IF bErrorBlinking THEN
	Error := FALSE;
END_IF

IF NOT Execute THEN
	bErrorBlinking := FALSE;
	tonErrorResetDelay.IN := FALSE;
	eSTATE:=STATE_RESETTING;
END_IF
END_METHOD

METHOD  M_STATE_EXECUTING
VAR_INPUT
END_VAR
VAR_INST
	bMoveConveyorForward : BOOL;
	bMoveConveyorBackrward : BOOL;
END_VAR

VAR
	bCylinderCheck : BOOL := TRUE;
END_VAR
Busy :=TRUE;
SensorOnConveyor := INPUT.bDifferentSizeCV_BoxDetect5_Sensor;

// ============================================================
// (A) Step 切換 → Timer 完整歸零 (Fix 1)
// ============================================================
IF uiExecutingStep <> uiExecutingStep_Last THEN
	tonTimeOut(IN:=FALSE);
	tonTimeDelay(IN:=FALSE);
	tonLeaveDebounce(IN:=FALSE);
	uiExecutingStep_Last := uiExecutingStep;
END_IF

// ============================================================
// (B) TurnTable Interlock (Fix 3)
// Place 下爪區間 (2200~2499) 與 TT 偵測區間 (2600) 期間
// TurnTable 不可移動 (pick 階段在 I5 conveyor,與 TT 無關)
// ============================================================
IF (uiExecutingStep >= 2200 AND uiExecutingStep <= 2499)
OR (uiExecutingStep = 2600)
THEN
	IF arAxisCtrl_gb[AxisNo.TurnTable].Admin.Axis.Status.Moving THEN
		_Error := TRUE;
		uiResumeStep := uiExecutingStep;
		strStatus := M_FormatManagedStatus(
			AlarmId := GVL_ErrorCode.GC_ALARM_ALC_OUTROBOT_EMPTY,
			InnerMessage := GVL_ErrorCode.GC_MSG_0174);
		Status := strStatus;
		Error := TRUE;
	END_IF
END_IF

// ============================================================
// (C) Pause 處理 (Fix 4) - 僅在「安全 step」生效
// ============================================================
bCanPause :=
	   uiExecutingStep = 0
	OR uiExecutingStep = 100
	OR uiExecutingStep = 200
	OR uiExecutingStep = 1000
	OR uiExecutingStep = 1100
	OR uiExecutingStep = 1400
	OR uiExecutingStep = 1900
	OR uiExecutingStep = 2000
	OR uiExecutingStep = 2100
	OR uiExecutingStep = 2500;

// Pause 釋放邊緣 → 強制 timer 歸零 (避免 release 瞬間誤判)
IF bPauseLast AND NOT Pause THEN
	tonTimeOut(IN:=FALSE);
	tonTimeDelay(IN:=FALSE);
	tonLeaveDebounce(IN:=FALSE);
END_IF
bPauseLast := Pause;

IF Pause AND bCanPause THEN
	bMoveConveyorForward := FALSE;
	bMoveConveyorBackrward := FALSE;
	IF __ISVALIDREF(ConveyorMotor) THEN
		ConveyorMotor.M_MotorStop();
	END_IF
	tonTimeOut(IN:=FALSE);
	tonTimeDelay(IN:=FALSE);
	tonLeaveDebounce(IN:=FALSE);
	Busy := TRUE;
	RETURN;
END_IF

// ============================================================
// Conveyor 連續控制 (沿用既有 latched flag)
// ============================================================
IF bMoveConveyorForward THEN
	IF NOT ConveyorMotor.InBackWard THEN
		ConveyorMotor.M_MoveForward();
	END_IF
END_IF
IF bMoveConveyorBackrward THEN
	IF NOT ConveyorMotor.InForWard THEN
		ConveyorMotor.M_MoveBackward();
	END_IF
END_IF

CASE uiExecutingStep OF

0: //Entry - VAR_INST reset + working conditions
	// VAR_INST 私有給本 method,DORMANT 看不到,必須在此 reset
	bMoveConveyorForward := FALSE;
	bMoveConveyorBackrward := FALSE;

	IF GVL_Machine.PackTags[UnitNo.Allocate].Status.UnitModeCurrent <> E_UnitMode.Auto THEN
		strStatus := 'Not in Auto mode';
		_UniqueErrorCode := 'E_NOT_AUTO_MODE';
		_Error := TRUE;
	ELSIF bResumeEnabled AND uiResumeStep > 0 THEN
		// 續做模式: M_GetWorkingConditions 重新取 clamping info (可能已改)
		IF M_GetWorkingConditions() THEN
			M_RecoveryAllObjects();
			// Safety: 若仍夾著箱,強制走 placing 流程 (絕不能回 pick 再抓一個)
			IF bClipHasBox[0] OR bClipHasBox[1] THEN
				IF bClipHasBox[0] THEN
					iWorkingIndex := 0;
				ELSE
					iWorkingIndex := 1;
				END_IF
				// 對齊 pick/place 進度: 未握箱的側視為「無須再處理」
				bPickedA := UseA;
				bPickedB := UseB;
				bPlacedA := UseA AND NOT bClipHasBox[0];
				bPlacedB := UseB AND NOT bClipHasBox[1];
				uiExecutingStep := 2000;	// 直接進 placing (會重檢 TT 角度)
			ELSE
				uiExecutingStep := M_GetResumeEntryStep(uiErrorStep:=uiResumeStep);
			END_IF
			bResumeEnabled := FALSE;
			uiResumeStep := 0;
		ELSE
			_Error := TRUE;
		END_IF
	ELSE
		// 正常啟動: DORMANT 已 reset 所有 FB-level flag,此處讀 input + recover 物件
		IF M_GetWorkingConditions() THEN
			M_RecoveryAllObjects();
			uiExecutingStep := 100;
		ELSE
			_Error := TRUE;
		END_IF
	END_IF

100: //Check command
	IF __ISVALIDREF(PressCylinderOnI5) THEN
		IF PressCylinderOnI5.xError THEN
			PressCylinderOnI5.M_Reset();
		ELSE
			PressCylinderOnI5.M_Retract();
		END_IF
	END_IF

	IF M_CheckCommand() THEN
		uiExecutingStep:=200;
	ELSE
		_Error := TRUE;
	END_IF

200: // Check no boxes on TurnTable (殘箱 → 不可續做)
	IF (UseA AND INPUT.bTurnTable_R1Detect_Sensor) OR (UseB AND INPUT.bTurnTable_R2Detect_Sensor) THEN
		_Abort:=TRUE;
		uiResumeStep := 0;	// 殘箱錯誤禁止續做
		strStatus := M_FormatManagedStatus(
			AlarmId := GVL_ErrorCode.GC_ALARM_ALC_OUTROBOT_EMPTY,
			InnerMessage := GVL_ErrorCode.GC_MSG_0012);
		Status := strStatus;
		Error := TRUE;
	ELSE
		IF UseA THEN
			iWorkingIndex :=0;
		ELSE
			iWorkingIndex :=1;
		END_IF
		uiExecutingStep:=1000;
	END_IF

1000: // Move conveyor forward + send OutRobot to picking pos
	bMoveConveyorForward:=TRUE;
	arAxisCtrl_gb[AxisNo.OutRobot_X].PosMode.Position := PickingPos[iWorkingIndex].X_Pos;
	arAxisCtrl_gb[AxisNo.OutRobot_Y].PosMode.Position := PickingPos[iWorkingIndex].Y_Pos;
	IF ConveyorMotor.InForWard THEN
		uiExecutingStep:=1100;
	END_IF

1100: // Wait box arriving sensor (1s debounce)
	tonTimeDelay(IN:=SensorOnConveyor, PT:=T#1S);
	IF tonTimeDelay.Q THEN
		uiExecutingStep:=1200;
	ELSE
		tonTimeOut(IN:=TRUE, PT:=T#15S);
		IF tonTimeOut.Q THEN
			_Abort := TRUE;
			uiResumeStep := uiExecutingStep;
			strStatus := M_FormatManagedStatus(
				AlarmId := GVL_ErrorCode.GC_ALARM_ALC_OUTROBOT_EMPTY,
				InnerMessage := GVL_ErrorCode.GC_MSG_0088);
			Status := strStatus;
			Error := TRUE;
		END_IF
	END_IF

1200: // (預留) Press second box - 目前不執行,直接 fall-through
	uiExecutingStep:=1300;

1300: // Stop conveyor
	ConveyorMotor.M_MotorStop();
	bMoveConveyorForward:=FALSE;
	bMoveConveyorBackrward:=FALSE;
	IF ConveyorMotor.InStopped THEN
		uiExecutingStep:=1400;
	END_IF

1400: // Wait OutRobot XY arrive (pick)
	IF (arAxisStatus_gb[AxisNo.OutRobot_X].Admin._OpModeAck = ModePosAbs AND arAxisStatus_gb[AxisNo.OutRobot_X].Admin.CmdDone)
	AND (arAxisStatus_gb[AxisNo.OutRobot_Y].Admin._OpModeAck = ModePosAbs AND arAxisStatus_gb[AxisNo.OutRobot_Y].Admin.CmdDone)
	THEN
		uiExecutingStep:=1500;
	ELSE
		tonTimeOut(IN:=TRUE, PT:=T#15S);
		IF tonTimeOut.Q THEN
			_Error := TRUE;
			uiResumeStep := uiExecutingStep;
			strStatus := M_FormatManagedStatus(
				AlarmId := GVL_ErrorCode.GC_ALARM_ALC_OUTROBOT_EMPTY,
				InnerMessage := GVL_ErrorCode.GC_MSG_0083);
			Status := strStatus;
			Error := TRUE;
		END_IF
	END_IF

1500: // Clip down (pick) - Fix 2: 下爪前位置再確認
	IF NOT M_IsOutRobotAtPos(TargetPos:=PickingPos[iWorkingIndex]) THEN
		_Error := TRUE;
		uiResumeStep := uiExecutingStep;
		strStatus := M_FormatManagedStatus(
			AlarmId := GVL_ErrorCode.GC_ALARM_ALC_OUTROBOT_EMPTY,
			InnerMessage := GVL_ErrorCode.GC_MSG_0172);
		Status := strStatus;
		Error := TRUE;
	ELSE
		// Sync 對稱化 (S1/S2): sync 時兩爪同動同檢查
		IF bSyncPick THEN
			Cylinders[0].M_Extend();
			Cylinders[1].M_Extend();
			bCylinderCheck := Cylinders[0].InFrontPosition AND Cylinders[1].InFrontPosition;
		ELSE
			Cylinders[iWorkingIndex].M_Extend();
			bCylinderCheck := Cylinders[iWorkingIndex].InFrontPosition;
		END_IF
		IF bCylinderCheck THEN
			uiExecutingStep:=1700;
		ELSE
			tonTimeOut(IN:=TRUE, PT:=T#15S);
			IF tonTimeOut.Q THEN
				_Abort := TRUE;
				uiResumeStep := uiExecutingStep;
				strStatus := M_FormatManagedStatus(
					AlarmId := GVL_ErrorCode.GC_ALARM_ALC_OUTROBOT_EMPTY,
					InnerMessage := GVL_ErrorCode.GC_MSG_0048);
				Status := strStatus;
				Error := TRUE;
			END_IF
		END_IF
	END_IF

1700: // Clip close (pick)
	IF bSyncPick THEN
		Clips[0].M_Extend();
		Clips[1].M_Extend();
		bCylinderCheck := Clips[0].InFrontPosition AND Clips[1].InFrontPosition;
	ELSE
		Clips[iWorkingIndex].M_Extend();
		bCylinderCheck := Clips[iWorkingIndex].InFrontPosition;
	END_IF
	IF bCylinderCheck THEN
		// Safety: 標記夾到箱 (sync 時兩爪都標)
		IF bSyncPick THEN
			bClipHasBox[0] := TRUE;
			bClipHasBox[1] := TRUE;
		ELSE
			bClipHasBox[iWorkingIndex] := TRUE;
		END_IF
		uiExecutingStep:=1800;
	ELSE
		tonTimeOut(IN:=TRUE, PT:=T#15S);
		IF tonTimeOut.Q THEN
			_Abort := TRUE;
			uiResumeStep := uiExecutingStep;
			strStatus := M_FormatManagedStatus(
				AlarmId := GVL_ErrorCode.GC_ALARM_ALC_OUTROBOT_EMPTY,
				InnerMessage := GVL_ErrorCode.GC_MSG_0026);
			Status := strStatus;
			Error := TRUE;
		END_IF
	END_IF

1800: // Clip up (pick)
	IF bSyncPick THEN
		Cylinders[0].M_Retract();
		Cylinders[1].M_Retract();
		bCylinderCheck := Cylinders[0].InRearPosition AND Cylinders[1].InRearPosition;
	ELSE
		Cylinders[iWorkingIndex].M_Retract();
		bCylinderCheck := Cylinders[iWorkingIndex].InRearPosition;
	END_IF
	IF bCylinderCheck THEN
		uiExecutingStep:=1850;
	ELSE
		tonTimeOut(IN:=TRUE, PT:=T#15S);
		IF tonTimeOut.Q THEN
			_Abort := TRUE;
			uiResumeStep := uiExecutingStep;
			strStatus := M_FormatManagedStatus(
				AlarmId := GVL_ErrorCode.GC_ALARM_ALC_OUTROBOT_EMPTY,
				InnerMessage := GVL_ErrorCode.GC_MSG_0050);
			Status := strStatus;
			Error := TRUE;
		END_IF
	END_IF

1850: // Confirm box left conveyor sensor
	// ============================================================
	// TEMP (2026-04-30): A、B 兩爪皆暫時跳過離開檢查
	// 原因: conveyor sensor (BoxDetect5) 只能反映 conveyor 上有無箱,
	//       無法保證箱真的被夾在爪上。A 原本就跳過 (避免上游補料壓
	//       sensor 誤判), B 因相同顧慮也暫時不檢查。
	// 復原條件: 爪上加裝 box-detect sensor,或上游補料時序確認後。
	// 復原方式: 移除本無條件跳過區塊,還原下方 (* *) 內的原邏輯。
	// ============================================================
	tonLeaveDebounce(IN:=FALSE, PT:=T#1S);
	tonTimeOut(IN:=FALSE, PT:=T#15S);
	IF __ISVALIDREF(PressCylinderOnI5) THEN
		PressCylinderOnI5.M_Retract();
	END_IF
	uiExecutingStep:=1900;

	(* ---- 原離開檢查邏輯 (TEMP 解除後恢復本段, 移除上方無條件跳過) ----
	// 若還有下一爪要夾,上游補料會壓住同一顆 sensor 造成誤判,直接跳過離開檢查
	IF NOT bSyncPick
		AND ( (iWorkingIndex = 0 AND UseB AND NOT bPickedB)
		   OR (iWorkingIndex = 1 AND UseA AND NOT bPickedA) )
	THEN
		tonLeaveDebounce(IN:=FALSE, PT:=T#1S);
		tonTimeOut(IN:=FALSE, PT:=T#15S);
		IF __ISVALIDREF(PressCylinderOnI5) THEN
			PressCylinderOnI5.M_Retract();
		END_IF
		uiExecutingStep:=1900;
	ELSE
		tonLeaveDebounce(IN:=NOT SensorOnConveyor, PT:=T#1S);
		IF tonLeaveDebounce.Q THEN
			IF __ISVALIDREF(PressCylinderOnI5) THEN
				PressCylinderOnI5.M_Retract();
			END_IF
			uiExecutingStep:=1900;
		ELSE
			tonTimeOut(IN:=TRUE, PT:=T#15S);
			IF tonTimeOut.Q THEN
				_Abort := TRUE;
				uiResumeStep := uiExecutingStep;
				strStatus := M_FormatManagedStatus(
					AlarmId := GVL_ErrorCode.GC_ALARM_ALC_OUTROBOT_EMPTY,
					InnerMessage := GVL_ErrorCode.GC_MSG_0015);
			END_IF
		END_IF
	END_IF
	*)

1900: // Next pick? (附加 bug fix: 用 bPickedA/B 旗標,避免 iWorkingIndex 漏放 B)
	IF bSyncPick THEN
		bPickedA := TRUE;
		bPickedB := TRUE;
	ELSIF iWorkingIndex = 0 THEN
		bPickedA := TRUE;
	ELSE
		bPickedB := TRUE;
	END_IF
	IF UseA AND NOT bPickedA THEN
		iWorkingIndex := 0;
		uiExecutingStep := 1000;
	ELSIF UseB AND NOT bPickedB THEN
		iWorkingIndex := 1;
		uiExecutingStep := 1000;
	ELSE
		// 全部 pick 完,進入 placing
		IF UseA THEN
			iWorkingIndex := 0;
		ELSE
			iWorkingIndex := 1;
		END_IF
		uiExecutingStep := 2000;
	END_IF

2000: // Move to placing pos - TurnTable 角度 gate
	IF NOT M_IsTurnTableAtPlaceAngle() THEN
		_Error := TRUE;
		uiResumeStep := uiExecutingStep;
		strStatus := M_FormatManagedStatus(
			AlarmId := GVL_ErrorCode.GC_ALARM_ALC_OUTROBOT_EMPTY,
			InnerMessage := GVL_ErrorCode.GC_MSG_0175);
		Status := strStatus;
		Error := TRUE;
	ELSE
		arAxisCtrl_gb[AxisNo.OutRobot_X].PosMode.Position := PlacingPos[iWorkingIndex].X_Pos;
		arAxisCtrl_gb[AxisNo.OutRobot_Y].PosMode.Position := PlacingPos[iWorkingIndex].Y_Pos;
		uiExecutingStep:=2100;
	END_IF

2100: // Wait OutRobot XY arrive (place) + TurnTable 靜止 (Fix 3 修正對象)
	IF (arAxisStatus_gb[AxisNo.OutRobot_X].Admin._OpModeAck = ModePosAbs AND arAxisStatus_gb[AxisNo.OutRobot_X].Admin.CmdDone)
	AND (arAxisStatus_gb[AxisNo.OutRobot_Y].Admin._OpModeAck = ModePosAbs AND arAxisStatus_gb[AxisNo.OutRobot_Y].Admin.CmdDone)
	AND NOT arAxisCtrl_gb[AxisNo.TurnTable].Admin.Axis.Status.Moving
	THEN
		uiExecutingStep:=2200;
	ELSE
		tonTimeOut(IN:=TRUE, PT:=T#15S);
		IF tonTimeOut.Q THEN
			_Error := TRUE;
			uiResumeStep := uiExecutingStep;
			strStatus := M_FormatManagedStatus(
				AlarmId := GVL_ErrorCode.GC_ALARM_ALC_OUTROBOT_EMPTY,
				InnerMessage := GVL_ErrorCode.GC_MSG_0084);
			Status := strStatus;
			Error := TRUE;
		END_IF
	END_IF

2200: // Clip down (place) - Fix 2: 下爪前位置再確認
	IF NOT M_IsOutRobotAtPos(TargetPos:=PlacingPos[iWorkingIndex]) THEN
		_Error := TRUE;
		uiResumeStep := uiExecutingStep;
		strStatus := M_FormatManagedStatus(
			AlarmId := GVL_ErrorCode.GC_ALARM_ALC_OUTROBOT_EMPTY,
			InnerMessage := GVL_ErrorCode.GC_MSG_0173);
		Status := strStatus;
		Error := TRUE;
	ELSE
		// Sync 對稱化 (S2): sync 時兩爪同動同檢查; 非 sync 只動 iWorkingIndex
		IF bSyncPlace THEN
			Cylinders[0].M_Extend();
			Cylinders[1].M_Extend();
			bCylinderCheck := Cylinders[0].InFrontPosition AND Cylinders[1].InFrontPosition;
		ELSE
			Cylinders[iWorkingIndex].M_Extend();
			bCylinderCheck := Cylinders[iWorkingIndex].InFrontPosition;
		END_IF
		IF bCylinderCheck THEN
			uiExecutingStep:=2300;
		ELSE
			tonTimeOut(IN:=TRUE, PT:=T#15S);
			IF tonTimeOut.Q THEN
				_Abort := TRUE;
				uiResumeStep := uiExecutingStep;
				strStatus := M_FormatManagedStatus(
					AlarmId := GVL_ErrorCode.GC_ALARM_ALC_OUTROBOT_EMPTY,
					InnerMessage := GVL_ErrorCode.GC_MSG_0051);
				Status := strStatus;
				Error := TRUE;
			END_IF
		END_IF
	END_IF

2300: // Clip open (place)
	IF bSyncPlace THEN
		Clips[0].M_Retract();
		Clips[1].M_Retract();
		bCylinderCheck := Clips[0].InRearPosition AND Clips[1].InRearPosition;
	ELSE
		Clips[iWorkingIndex].M_Retract();
		bCylinderCheck := Clips[iWorkingIndex].InRearPosition;
	END_IF
	IF bCylinderCheck THEN
		// Safety: 箱已放下 (sync 時兩爪都清,S4)
		IF bSyncPlace THEN
			bClipHasBox[0] := FALSE;
			bClipHasBox[1] := FALSE;
		ELSE
			bClipHasBox[iWorkingIndex] := FALSE;
		END_IF
		uiExecutingStep:=2400;
	ELSE
		tonTimeOut(IN:=TRUE, PT:=T#15S);
		IF tonTimeOut.Q THEN
			_Abort := TRUE;
			uiResumeStep := uiExecutingStep;
			strStatus := M_FormatManagedStatus(
				AlarmId := GVL_ErrorCode.GC_ALARM_ALC_OUTROBOT_EMPTY,
				InnerMessage := GVL_ErrorCode.GC_MSG_0027);
			Status := strStatus;
			Error := TRUE;
		END_IF
	END_IF

2400: // Clip up (place)
	IF bSyncPlace THEN
		Cylinders[0].M_Retract();
		Cylinders[1].M_Retract();
		bCylinderCheck := Cylinders[0].InRearPosition AND Cylinders[1].InRearPosition;
	ELSE
		Cylinders[iWorkingIndex].M_Retract();
		bCylinderCheck := Cylinders[iWorkingIndex].InRearPosition;
	END_IF
	IF bCylinderCheck THEN
		uiExecutingStep:=2500;
	ELSE
		tonTimeOut(IN:=TRUE, PT:=T#15S);
		IF tonTimeOut.Q THEN
			_Abort := TRUE;
			uiResumeStep := uiExecutingStep;
			strStatus := M_FormatManagedStatus(
				AlarmId := GVL_ErrorCode.GC_ALARM_ALC_OUTROBOT_EMPTY,
				InnerMessage := GVL_ErrorCode.GC_MSG_0053);
			Status := strStatus;
			Error := TRUE;
		END_IF
	END_IF

2500: // Next place? (附加 bug fix: 用 bPlacedA/B 旗標)
	IF bSyncPlace THEN
		bPlacedA := TRUE;
		bPlacedB := TRUE;
	ELSIF iWorkingIndex = 0 THEN
		bPlacedA := TRUE;
	ELSE
		bPlacedB := TRUE;
	END_IF
	IF UseA AND NOT bPlacedA THEN
		iWorkingIndex := 0;
		uiExecutingStep := 2000;
	ELSIF UseB AND NOT bPlacedB THEN
		iWorkingIndex := 1;
		uiExecutingStep := 2000;
	ELSE
		uiExecutingStep := 2600;
	END_IF

2600: // Check box on TurnTable (沒放好 → 不可續做)
	IF (UseA AND NOT INPUT.bTurnTable_R1Detect_Sensor) OR (UseB AND NOT INPUT.bTurnTable_R2Detect_Sensor) THEN
		_Error:=TRUE;
		uiResumeStep := 0;	// 沒放好 → 禁止續做,需人員處理
		strStatus := M_FormatManagedStatus(
			AlarmId := GVL_ErrorCode.GC_ALARM_ALC_OUTROBOT_EMPTY,
			InnerMessage := GVL_ErrorCode.GC_MSG_0008);
		Status := strStatus;
		Error := TRUE;
	ELSE
		uiExecutingStep:=3000;
	END_IF

3000: // Finish
	bMoveConveyorForward:=FALSE;
	bMoveConveyorBackrward:=FALSE;
	_Executed:=TRUE;

END_CASE

IF NOT Execute THEN
	eState:=STATE_RESETTING;
END_IF
IF _Error THEN
	eState:=STATE_ERROR;
END_IF
IF _Abort THEN
	eSTATE:=STATE_ABORTING;
END_IF
IF _Executed THEN
	eSTATE:=STATE_Done;
END_IF
END_METHOD

METHOD  M_STATE_RESETTING
VAR_INPUT
END_VAR
Busy := TRUE;
Error := _Error;

// Timer 確保歸零 (避免 RESET→DORMANT→EXECUTING 殘留)
tonTimeOut(IN:=FALSE);
tonTimeDelay(IN:=FALSE);
tonLeaveDebounce(IN:=FALSE);

CASE uiResettingStep OF

	0:

		IF __ISVALIDREF(ConveyorMotor) THEN
			ConveyorMotor.M_MotorStop();
		END_IF
		M_RecoveryAllObjects();
		IF __ISVALIDREF(PressCylinderOnI5) THEN
			IF PressCylinderOnI5.xError THEN
				PressCylinderOnI5.M_Reset();
			ELSE
				PressCylinderOnI5.M_Retract();
			END_IF
		END_IF
		uiResettingStep:=9999;

	9999:
		Done := FALSE;
		Busy := FALSE;
		_ResetCompleted:=TRUE;
END_CASE
IF _ResetCompleted THEN
	eSTATE:=STATE_DORMANT;
END_IF
END_METHOD

END_FUNCTION_BLOCK

// ---- Library/20_MachineUnits/22_AllocateArea/Service/FB_OutRobot_RareBoxMove.TcPOU
FUNCTION_BLOCK FB_OutRobot_RareBoxMove EXTENDS FB_ObjectBase_V2
VAR_INPUT
//    Execute    :BOOL;   // True : This prog will start.
//    Abort      :BOOL;   // True : This prog will be abort.
//    Reset      :BOOL;   // True : This prog will be reset.
//    ObjectName :STRING; // Set this fb name(About it's action)
	INPUT            			   : REFERENCE TO ST_InputTable;	
	Cylinder   					   : REFERENCE TO UNI_CylinderList;
	Motor      					   : REFERENCE TO UNI_MotorList;
	Cylinders					   : REFERENCE TO ARRAY[0..1] OF FB_Cylinder;
	Clips						   : REFERENCE TO ARRAY[0..1] OF FB_Cylinder;
	AutoMode_OutRobotMoveMove : st_AutoMode_ClampingBoxesJob;	
END_VAR

VAR_OUTPUT
//    Busy    :BOOL;        // True : This prog is running.
//    Done    :BOOL;        // True : Command has been executed.
//    Aborted :BOOL;        // True : This prog is aborted.
//    Error   :BOOL;        // True : This prog has an error.
//    ErrorID :UINT;       // Output ErrorID
//    Status  :T_MaxString; // Output this prog status by string(255bytes)
END_VAR

VAR
//    eState :E_MethodStatus_Basic;
//	uiExecutingStep : UDINT; // This var is used to been controll STATE_EXECUTING process.
//	uiResettingStep : UDINT;
//	uiAbortingStep : UDINT;
//	_Executed :BOOL; // Executing process completed.
//	_Error : BOOL; // FB has an error.
//	_ResetCompleted : BOOL; // FB resetting completed.
//	_AbortCompleted : BOOL; // FB aborting completed.
//	_Abort		: BOOL;
	strStatus	: STRING;
	uiResumeStep : UDINT;
	tonTimeOut   :TON;
	tonTimeDelay   :TON;
	tonLeaveDebounce : TON;	// 1600 等箱離開 R sensor 去抖
	iWorkingIndex : INT;
	_UniqueErrorCode :STRING;
	PickingPos	: ARRAY[0..1] OF ST_PositionTable;
	PlacingPos  : ARRAY[0..1] OF ST_PositionTable;
	bSyncPick	: BOOL;
	bSyncPlace	: BOOL;
	SensorOnConveyor			   : BIT;
	ConveyorMotor				   : REFERENCE TO FB_Motor;
	UseA	: BOOL;
	UseB	: BOOL;
	bMotorMoveForward : BOOL;
	lrEpsPos 	: LREAL := 0.001;	// 浮點座標比較容差 (sync 判斷用)
	// Step 切換偵測 (timer 乾淨重置)
	uiExecutingStep_Last : UDINT;
	// Resume / Pause 機制
	bResumeEnabled : BOOL;
	bCanPause : BOOL;
	bPauseLast : BOOL;
	trigErrorReset : R_TRIG;
	tonErrorResetDelay : TON;
	bErrorBlinking : BOOL;
	// 雙 clip pick / place 旗標 (取代易誤的 iWorkingIndex 共用)
	bPickedA : BOOL;
	bPickedB : BOOL;
	bPlacedA : BOOL;
	bPlacedB : BOOL;
	// Safety: 夾爪是否正夾著箱 (latched, 1300 閉夾→TRUE, 2300 開夾→FALSE)
	bClipHasBox : ARRAY[0..1] OF BOOL;
	
	_bRetry  : BOOL;
END_VAR

A00_BasicUnits();
SUPER^.A10_StateControl();

ACTION A00_BasicUnits:
// Timer 由各 step 自行呼叫並傳 IN/PT,此處不做 freerun call,
// 避免「IN 殘留 TRUE」造成 step 切換後 timer 不歸零。
END_ACTION

METHOD GetModelState
VAR_OUTPUT
    xDone    :BOOL;
    xBusy    :BOOL;
    xError   :BOOL;
    xAborted :BOOL;
    iErrorID :UDINT;
	UniqueErrorCode : STRING;
END_VAR
xDone    := Done;
xBusy    := Busy;
xError   := Error;
xAborted := Aborted;
iErrorID := ErrorID;
UniqueErrorCode := THIS^.UniqueErrorCode;
END_METHOD

METHOD GetName : STRING
GetName := ObjectName;
END_METHOD

METHOD PRIVATE M_CheckCommand : BOOL
VAR_INPUT
END_VAR
IF NOT AutoMode_OutRobotMoveMove.ClampingInfo.UseClibA AND NOT AutoMode_OutRobotMoveMove.ClampingInfo.UseClibB THEN
	M_CheckCommand := FALSE;
	strStatus 	   := 'FB_OutRobot_RareBoxMove , Wrong Command Neither Clamp was used';
	RETURN;
END_IF
IF AutoMode_OutRobotMoveMove.ClampingInfo.TargetOfClipA <> AutoMode_OutRobotMoveMove.ClampingInfo.TargetOfClipB THEN
	M_CheckCommand := FALSE;
	strStatus 	   := 'FB_OutRobot_RareBoxMove , Wrong Command ClampA,B need same TargetPos';
	RETURN;
END_IF

M_CheckCommand:=true;
END_METHOD

METHOD PRIVATE M_GetResumeEntryStep : UDINT
VAR_INPUT
	uiErrorStep : UDINT;
END_VAR
// Resume 入口對照表: 錯誤點 → 重新進入的安全 checkpoint
CASE uiErrorStep OF
	1000, 1100:
		M_GetResumeEntryStep := 1000;	// 重發 XY 指令
	1200, 1300, 1400, 1500, 1600:
		M_GetResumeEntryStep := 1000;	// pick 階段錯誤 → 重發 XY 從頭 pick
	2000, 2100, 2150:
		M_GetResumeEntryStep := 2000;	// 重發 XY + conveyor
	2200, 2300, 2400, 2500:
		M_GetResumeEntryStep := 2000;	// place 階段錯誤 → 重發 XY 從頭 place
	2600, 2700:
		M_GetResumeEntryStep := 2600;	// conveyor handoff 重做
ELSE
	M_GetResumeEntryStep := 0;	// fallback
END_CASE
END_METHOD

METHOD PRIVATE M_GetWorkingConditions : BOOL
VAR_INPUT
END_VAR
//For rare box move , Boxes must place on same position , therefor only work with TargetPosition of ClipA

IF AutoMode_OutRobotMoveMove.ClampingInfo.TargetOfClipA = 5 THEN	
	ConveyorMotor REF= Motor.List.TransmitDifferentSideCV;
ELSIF AutoMode_OutRobotMoveMove.ClampingInfo.TargetOfClipA = 6 THEN
	ConveyorMotor REF= Motor.List.TransmitSameSideCV;
ELSIF AutoMode_OutRobotMoveMove.ClampingInfo.TargetOfClipA = 3 THEN
	ConveyorMotor REF= Motor.List.TransmitDifferentSideCV;
ELSIF AutoMode_OutRobotMoveMove.ClampingInfo.TargetOfClipA = 4 THEN
	ConveyorMotor REF= Motor.List.TransmitSameSideCV;	
END_IF

IF AutoMode_OutRobotMoveMove.ClampingInfo.TargetOfClipA=5 OR AutoMode_OutRobotMoveMove.ClampingInfo.TargetOfClipA=6 THEN
		bMotorMoveForward := FALSE;
	ELSE
		bMotorMoveForward := TRUE;	
END_IF
IF AutoMode_OutRobotMoveMove.ClampingInfo.UseClibA THEN
	PickingPos[0] :=FUN_GetPositionTableData('R',1,0);
	UseA := TRUE;
	CASE  AutoMode_OutRobotMoveMove.ClampingInfo.TargetOfClipA OF	
		
	3,4:
		PlacingPos[0] :=FUN_GetPositionTableData('O',AutoMode_OutRobotMoveMove.ClampingInfo.TargetOfClipA,0);
	5,6:
		PlacingPos[0] :=FUN_GetPositionTableData('I',AutoMode_OutRobotMoveMove.ClampingInfo.TargetOfClipA,0);
	ELSE
		strStatus := M_FormatManagedStatus(
			AlarmId := GVL_ErrorCode.GC_ALARM_ALC_OUTROBOT_RARE,
			InnerMessage := GVL_ErrorCode.GC_MSG_0157);
		Status := strStatus;
		Error := TRUE;
		M_GetWorkingConditions := FALSE;
		RETURN;
	END_CASE
END_IF

IF AutoMode_OutRobotMoveMove.ClampingInfo.UseClibB THEN
	PickingPos[1] :=FUN_GetPositionTableData('R',2,1);
	UseB :=TRUE;
	CASE AutoMode_OutRobotMoveMove.ClampingInfo.TargetOfClipA OF
		
	3,4:
		PlacingPos[1] :=FUN_GetPositionTableData('O',AutoMode_OutRobotMoveMove.ClampingInfo.TargetOfClipA,1);
	5,6 :
		PlacingPos[1] :=FUN_GetPositionTableData('I',AutoMode_OutRobotMoveMove.ClampingInfo.TargetOfClipA,1);
	ELSE
		strStatus := M_FormatManagedStatus(
			AlarmId := GVL_ErrorCode.GC_ALARM_ALC_OUTROBOT_RARE,
			InnerMessage := GVL_ErrorCode.GC_MSG_0158);
		Status := strStatus;
		Error := TRUE;
		M_GetWorkingConditions := FALSE;
		RETURN;
	END_CASE
END_IF

// Sync 判斷一律用浮點容差 (lrEpsPos),避免 LREAL 直接比較被微誤差誤判
bSyncPick := UseA AND UseB
	AND ABS(PickingPos[0].X_Pos - PickingPos[1].X_Pos) < lrEpsPos
	AND ABS(PickingPos[0].Y_Pos - PickingPos[1].Y_Pos) < lrEpsPos;

bSyncPlace := UseA AND UseB
	AND ABS(PlacingPos[0].X_Pos - PlacingPos[1].X_Pos) < lrEpsPos
	AND ABS(PlacingPos[0].Y_Pos - PlacingPos[1].Y_Pos) < lrEpsPos;

M_GetWorkingConditions :=TRUE;
END_METHOD

METHOD PRIVATE M_IsOutRobotAtPos : BOOL
VAR_INPUT
	TargetPos : ST_PositionTable;
END_VAR
VAR
	lTol : LREAL := 0.1;
END_VAR
//lTol := GVL_HMI.Setup.Mechanical.OutRobotPositionTolerance;

M_IsOutRobotAtPos :=
		NOT arAxisCtrl_gb[AxisNo.OutRobot_X].Admin.Axis.Status.Moving
	AND NOT arAxisCtrl_gb[AxisNo.OutRobot_Y].Admin.Axis.Status.Moving
	AND ABS(arAxisCtrl_gb[AxisNo.OutRobot_X].Admin.Axis.NcToPlc.ActPos - TargetPos.X_Pos) <  0.1
	AND ABS(arAxisCtrl_gb[AxisNo.OutRobot_Y].Admin.Axis.NcToPlc.ActPos - TargetPos.Y_Pos) <  0.1;
END_METHOD

METHOD PRIVATE M_IsTurnTableAtStation : BOOL
VAR
	lActPos : LREAL;
	lTol    : LREAL := 0.1;
END_VAR
// Pick 前 TurnTable 必須位於 0/90/180/270/360 (任一 station)
// 使用 ModuloActPos 避免累積角度造成誤判
lActPos := ABS(arAxisCtrl_gb[AxisNo.TurnTable].Admin.Axis.NcToPlc.ModuloActPos);

M_IsTurnTableAtStation :=
	   FUN_CheckInPos(ActPos:=lActPos, TargetPos:=0,   ToleranceRange:=lTol)
	OR FUN_CheckInPos(ActPos:=lActPos, TargetPos:=90,  ToleranceRange:=lTol)
	OR FUN_CheckInPos(ActPos:=lActPos, TargetPos:=180, ToleranceRange:=lTol)
	OR FUN_CheckInPos(ActPos:=lActPos, TargetPos:=270, ToleranceRange:=lTol)
	OR FUN_CheckInPos(ActPos:=lActPos, TargetPos:=360, ToleranceRange:=lTol);
END_METHOD

METHOD PRIVATE M_RecoveryAllObjects : BOOL
VAR_INPUT
END_VAR
VAR 
	i : INT;
END_VAR
FOR i:=0 TO 1 DO
	// Clip: 有箱時絕對不張開 (safety),只清錯
	IF Clips[i].xError THEN
		Clips[i].M_Reset();
	ELSIF NOT bClipHasBox[i] THEN
		Clips[i].M_Retract();
	END_IF
	// Cylinder: 一律抬起 (空爪或有箱都安全)
	IF Cylinders[i].xError THEN
		Cylinders[i].M_Reset();
	ELSE
		Cylinders[i].M_Retract();
	END_IF
END_FOR

IF arAxisCtrl_gb[AxisNo.OutRobot_X].Admin.Axis.Status.Error THEN

	arAxisCtrl_gb[AxisNo.OutRobot_X].Admin.ClearError:= TRUE;
ELSE
	arAxisCtrl_gb[AxisNo.OutRobot_X].Admin.ClearError:= FALSE;
END_IF

IF arAxisCtrl_gb[AxisNo.OutRobot_Y].Admin.Axis.Status.Error THEN

	arAxisCtrl_gb[AxisNo.OutRobot_Y].Admin.ClearError:= TRUE;
ELSE
	arAxisCtrl_gb[AxisNo.OutRobot_Y].Admin.ClearError:= FALSE;
END_IF
END_METHOD

METHOD PRIVATE M_SensorUpdate : BOOL
VAR_INPUT
END_VAR
IF AutoMode_OutRobotMoveMove.ClampingInfo.TargetOfClipA = 5 THEN
	SensorOnConveyor := INPUT.bDifferentSizeCV_BoxDetect5_Sensor;
ELSIF AutoMode_OutRobotMoveMove.ClampingInfo.TargetOfClipA = 6 THEN
	SensorOnConveyor := INPUT.bSameSizeCV_BoxDetect5_Sensor;
ELSIF AutoMode_OutRobotMoveMove.ClampingInfo.TargetOfClipA = 3 THEN
	SensorOnConveyor := INPUT.bDifferentSizeCV_BoxDetect4_Sensor;
ELSIF AutoMode_OutRobotMoveMove.ClampingInfo.TargetOfClipA = 4 THEN
	SensorOnConveyor := INPUT.bSameSizeCV_BoxDetect4_Sensor;	
END_IF
END_METHOD

METHOD  M_STATE_ABORTED
VAR_INPUT
END_VAR
IF NOT _bRetry THEN
	ERROR 			:= TRUE;
	Busy    		:= FALSE;
	Aborted 		:= TRUE;
	Status 			:= strStatus;
	uiAbortingStep  := 0;
	_AbortCompleted := TRUE;
END_IF

IF reset THEN
	ERROR 	:= FALSE;
	Aborted := FALSE;
	_bRetry	:= TRUE;
END_IF

IF NOT Execute THEN
	eSTATE:=STATE_RESETTING;

// 續做: Reset+Execute 時設旗標,EXECUTING step 0 會跳到 ResumeStep
ELSIF Execute AND _bRetry AND uiResumeStep > 0 THEN
	Status  := '';
	bResumeEnabled := TRUE;
	uiExecutingStep := 0;
	eSTATE:=STATE_EXECUTING;
ELSIF Execute AND _bRetry AND uiResumeStep = 0 THEN
	strStatus := 'FB_OutRobot_RareBoxMove, this Error can not retry';
	eSTATE := STATE_ERROR;
END_IF
END_METHOD

METHOD  M_STATE_ABORTING
VAR_INPUT
END_VAR
VAR	
	i : INT;
	bCylinderCheck : BOOL :=true;
END_VAR
Error := TRUE;

// Timer 歸零
tonTimeOut(IN:=FALSE);
tonTimeDelay(IN:=FALSE);
tonLeaveDebounce(IN:=FALSE);

CASE uiAbortingStep OF
	0 :
		_Abort := FALSE;
		_bRetry := FALSE;
		IF __ISVALIDREF(ConveyorMotor) THEN
			ConveyorMotor.M_MotorStop();
		END_IF
		bCylinderCheck := TRUE;

		// Safety: 有箱的 clip 絕對不張開
		FOR i :=0 TO 1 DO
			IF Clips[i].xError THEN
				Clips[i].M_Reset();
			ELSIF NOT bClipHasBox[i] THEN
				Clips[i].M_Retract();
			END_IF
		END_FOR

		// Cylinder 一律抬起 (空爪或有箱都安全)
		FOR i :=0 TO 1 DO
			IF Cylinders[i].xError THEN
				Cylinders[i].M_Reset();
			END_IF
			Cylinders[i].M_Retract();
			bCylinderCheck:=bCylinderCheck AND Cylinders[i].InRearPosition;
		END_FOR

		IF bCylinderCheck THEN
			uiAbortingStep:=9999;
		END_IF
	9999:
		_Abort := FALSE;
		_AbortCompleted:=TRUE;
END_CASE

IF NOT Execute THEN
	eState := STATE_RESETTING;
ELSIF Execute AND _AbortCompleted THEN
	eSTATE :=STATE_ABORTED;
END_IF
END_METHOD

METHOD  M_STATE_DONE
VAR_INPUT
END_VAR
Busy 	:= FALSE;
Done	:=TRUE;

IF NOT Execute THEN
	eSTATE:=STATE_RESETTING;
END_IF
END_METHOD

METHOD  M_STATE_DORMANT
VAR_INPUT
END_VAR
Busy            := FALSE;
Done            := FALSE;
Aborted         := FALSE;
Error           := FALSE;
ErrorID         := 0;
Status          := '';
_ResetCompleted := FALSE;
_Error          := FALSE;
_Executed       := FALSE;
_Abort          := FALSE;
strStatus := M_FormatManagedStatus(
	AlarmId := GVL_ErrorCode.GC_ALARM_ALC_OUTROBOT_RARE,
	InnerMessage := GVL_ErrorCode.GC_MSG_0089);
Status := '';
Error := FALSE;
uiExecutingStep :=uiResettingStep :=0;
// Timer 完整歸零 (用實際 FB call,不是只設屬性)
tonTimeOut(IN:=FALSE);
tonTimeDelay(IN:=FALSE);
tonLeaveDebounce(IN:=FALSE);
uiExecutingStep_Last := 0;
_UniqueErrorCode:='0';
iWorkingIndex :=0;
bSyncPick := FALSE;
bSyncPlace := FALSE;
UseA := FALSE;
UseB := FALSE;
bMotorMoveForward := FALSE;
bPickedA := FALSE;
bPickedB := FALSE;
bPlacedA := FALSE;
bPlacedB := FALSE;
bPauseLast := FALSE;
bCanPause := FALSE;
_bRetry := FALSE;
_AbortCompleted := FALSE;
uiAbortingStep := 0;
bErrorBlinking := FALSE;
tonErrorResetDelay.IN := FALSE;
// 非續做模式才清 ResumeStep 與 ClipHasBox
IF NOT bResumeEnabled THEN
	uiResumeStep := 0;
	bClipHasBox[0] := FALSE;
	bClipHasBox[1] := FALSE;
END_IF
// 註: M_RecoveryAllObjects 不放 DORMANT 避免與其他 FB 搶 ClearError,
// 以及避免清掉 bClipHasBox 後誤張爪掉箱。僅 EXECUTING step 0 / RESETTING 呼叫。

IF Execute THEN
	eSTATE:=STATE_EXECUTING;
END_IF
END_METHOD

METHOD  M_STATE_ERROR
VAR_INPUT
END_VAR
ERROR   :=TRUE;
Busy	:=FALSE;
_Error  := FALSE;
Status := strStatus;
IF __ISVALIDREF(ConveyorMotor) THEN
	ConveyorMotor.M_MotorStop();
END_IF

// Reset 上升緣觸發 1 秒 Error 暫滅，之後重新亮回
trigErrorReset(CLK := reset);
IF trigErrorReset.Q THEN
	bErrorBlinking := TRUE;
END_IF

tonErrorResetDelay(IN := bErrorBlinking, PT := T#1S);
IF tonErrorResetDelay.Q THEN
	bErrorBlinking := FALSE;
END_IF

IF bErrorBlinking THEN
	Error := FALSE;
END_IF

IF NOT Execute THEN
	bErrorBlinking := FALSE;
	tonErrorResetDelay.IN := FALSE;
	eSTATE:=STATE_RESETTING;
END_IF
END_METHOD

METHOD  M_STATE_EXECUTING
VAR_INPUT
END_VAR
VAR_INST
	bMoveConveyorForward : BOOL;
	bMoveConveyorBackrward : BOOL;

END_VAR

VAR
	bCylinderCheck : BOOL := TRUE;
END_VAR
Busy :=TRUE;
M_SensorUpdate();

// ============================================================
// (A) Step 切換 → Timer 完整歸零 (Fix 1)
// ============================================================
IF uiExecutingStep <> uiExecutingStep_Last THEN
	tonTimeOut(IN:=FALSE);
	tonTimeDelay(IN:=FALSE);
	tonLeaveDebounce(IN:=FALSE);
	uiExecutingStep_Last := uiExecutingStep;
END_IF

// ============================================================
// (B) TurnTable Interlock (Fix 3)
// Pick 下爪區間 (1200~1499) 與 R 偵測區間 (1600) 期間
// TurnTable 不可移動 (place 階段在 conveyor,與 TT 無關)
// ============================================================
IF (uiExecutingStep >= 1200 AND uiExecutingStep <= 1499)
OR (uiExecutingStep = 1600)
THEN
	IF arAxisCtrl_gb[AxisNo.TurnTable].Admin.Axis.Status.Moving THEN
		_Error := TRUE;
		uiResumeStep := uiExecutingStep;
		strStatus := M_FormatManagedStatus(
			AlarmId := GVL_ErrorCode.GC_ALARM_ALC_OUTROBOT_RARE,
			InnerMessage := GVL_ErrorCode.GC_MSG_0174);
		Status := strStatus;
		Error := TRUE;
	END_IF
END_IF

// ============================================================
// (C) Pause 處理 (Fix 4) - 僅在「安全 step」生效
// ============================================================
bCanPause :=
	   uiExecutingStep = 0
	OR uiExecutingStep = 100
	OR uiExecutingStep = 200
	OR uiExecutingStep = 1000
	OR uiExecutingStep = 1100
	OR uiExecutingStep = 1500
	OR uiExecutingStep = 2000
	OR uiExecutingStep = 2100
	OR uiExecutingStep = 2150
	OR uiExecutingStep = 2500
	OR uiExecutingStep = 2700;

// Pause 釋放邊緣 → 強制 timer 歸零
IF bPauseLast AND NOT Pause THEN
	tonTimeOut(IN:=FALSE);
	tonTimeDelay(IN:=FALSE);
	tonLeaveDebounce(IN:=FALSE);
END_IF
bPauseLast := Pause;

IF Pause AND bCanPause THEN
	bMoveConveyorForward := FALSE;
	bMoveConveyorBackrward := FALSE;
	IF __ISVALIDREF(ConveyorMotor) THEN
		ConveyorMotor.M_MotorStop();
	END_IF
	tonTimeOut(IN:=FALSE);
	tonTimeDelay(IN:=FALSE);
	tonLeaveDebounce(IN:=FALSE);
	Busy := TRUE;
	RETURN;
END_IF

// ============================================================
// Conveyor 連續控制 (沿用既有 latched flag)
// ============================================================
IF bMoveConveyorForward THEN
	IF NOT ConveyorMotor.InBackWard THEN
		ConveyorMotor.M_MoveForward();
	END_IF
END_IF

IF bMoveConveyorBackrward THEN
	IF NOT ConveyorMotor.InForWard THEN
		ConveyorMotor.M_MoveBackward();
	END_IF
END_IF

CASE uiExecutingStep OF

0: //Entry - VAR_INST reset + 流程分流
	// VAR_INST 私有給本 method,DORMANT 看不到,必須在此 reset
	bMoveConveyorForward := FALSE;
	bMoveConveyorBackrward := FALSE;

	IF GVL_Machine.PackTags[UnitNo.Allocate].Status.UnitModeCurrent <> E_UnitMode.Auto THEN
		strStatus := 'Not in Auto mode';
		_UniqueErrorCode := 'E_NOT_AUTO_MODE';
		_Error := TRUE;
	ELSIF bResumeEnabled AND uiResumeStep > 0 THEN
		// 續做模式: M_GetWorkingConditions 重新取 input
		IF M_GetWorkingConditions() THEN
			M_RecoveryAllObjects();
			// Safety: 若仍夾著箱,強制走 placing 流程 (絕不能回 pick 再抓)
			IF bClipHasBox[0] OR bClipHasBox[1] THEN
				IF bClipHasBox[0] THEN
					iWorkingIndex := 0;
				ELSE
					iWorkingIndex := 1;
				END_IF
				bPickedA := UseA;
				bPickedB := UseB;
				bPlacedA := UseA AND NOT bClipHasBox[0];
				bPlacedB := UseB AND NOT bClipHasBox[1];
				uiExecutingStep := 2000;
			ELSE
				uiExecutingStep := M_GetResumeEntryStep(uiErrorStep:=uiResumeStep);
			END_IF
			bResumeEnabled := FALSE;
			uiResumeStep := 0;
		ELSE
			_Error := TRUE;
		END_IF
	ELSE
		// 正常啟動: DORMANT 已 reset 所有 FB-level flag,此處讀 input + recover 物件
		IF M_GetWorkingConditions() THEN
			M_RecoveryAllObjects();
			uiExecutingStep := 100;
		ELSE
			_Error := TRUE;
		END_IF
	END_IF

100: //Check command (M_GetWorkingConditions 已於 step 0 跑過)
	IF M_CheckCommand() THEN
		uiExecutingStep:=200;
	ELSE
		_Error :=TRUE;
	END_IF

200: // Check TT angle gate + 確認 R 上有箱
	IF NOT M_IsTurnTableAtStation() THEN
		_Abort := TRUE;
		uiResumeStep := uiExecutingStep;
		strStatus := M_FormatManagedStatus(
			AlarmId := GVL_ErrorCode.GC_ALARM_ALC_OUTROBOT_RARE,
			InnerMessage := GVL_ErrorCode.GC_MSG_0175);
		Status := strStatus;
		Error := TRUE;
	ELSIF (UseA AND NOT INPUT.bTurnTable_R1Detect_Sensor) OR (UseB AND NOT INPUT.bTurnTable_R2Detect_Sensor) THEN
		_Abort:=TRUE;
		uiResumeStep := 0;	// 沒箱可抓 → 不可續做
		strStatus := M_FormatManagedStatus(
			AlarmId := GVL_ErrorCode.GC_ALARM_ALC_OUTROBOT_RARE,
			InnerMessage := GVL_ErrorCode.GC_MSG_0009);
	ELSE
		IF UseA THEN
			iWorkingIndex :=0;
		ELSE
			iWorkingIndex :=1;
		END_IF
		uiExecutingStep:=1000;
	END_IF

1000: // Move OutRobot to picking pos (TurnTable R)
	arAxisCtrl_gb[AxisNo.OutRobot_X].PosMode.Position := PickingPos[iWorkingIndex].X_Pos;
	arAxisCtrl_gb[AxisNo.OutRobot_Y].PosMode.Position := PickingPos[iWorkingIndex].Y_Pos;
	uiExecutingStep:=1100;

1100: // Wait OutRobot XY arrive (pick on TT)
	IF (arAxisStatus_gb[AxisNo.OutRobot_X].Admin._OpModeAck = ModePosAbs AND arAxisStatus_gb[AxisNo.OutRobot_X].Admin.CmdDone)
	AND (arAxisStatus_gb[AxisNo.OutRobot_Y].Admin._OpModeAck = ModePosAbs AND arAxisStatus_gb[AxisNo.OutRobot_Y].Admin.CmdDone)
	AND NOT arAxisCtrl_gb[AxisNo.TurnTable].Admin.Axis.Status.Moving
	THEN
		uiExecutingStep:=1200;
	ELSE
		tonTimeOut(IN:=TRUE, PT:=T#15S);
		IF tonTimeOut.Q THEN
			_Abort := TRUE;
			uiResumeStep := uiExecutingStep;
			strStatus := M_FormatManagedStatus(
				AlarmId := GVL_ErrorCode.GC_ALARM_ALC_OUTROBOT_RARE,
				InnerMessage := GVL_ErrorCode.GC_MSG_0128);
		END_IF
	END_IF

1200: // Clip down (pick) - Fix 2: 下爪前位置再確認
	IF NOT M_IsOutRobotAtPos(TargetPos:=PickingPos[iWorkingIndex]) THEN
		_Abort := TRUE;
		uiResumeStep := uiExecutingStep;
		strStatus := M_FormatManagedStatus(
			AlarmId := GVL_ErrorCode.GC_ALARM_ALC_OUTROBOT_RARE,
			InnerMessage := GVL_ErrorCode.GC_MSG_0172);
		Status := strStatus;
		Error := TRUE;
	ELSE
		// Sync 對稱化 (S2): sync 時兩爪同動同檢查; 非 sync 只動 iWorkingIndex
		IF bSyncPick THEN
			Cylinders[0].M_Extend();
			Cylinders[1].M_Extend();
			bCylinderCheck := Cylinders[0].InFrontPosition AND Cylinders[1].InFrontPosition;
		ELSE
			Cylinders[iWorkingIndex].M_Extend();
			bCylinderCheck := Cylinders[iWorkingIndex].InFrontPosition;
		END_IF
		IF bCylinderCheck THEN
			uiExecutingStep:=1300;
		ELSE
			tonTimeOut(IN:=TRUE, PT:=T#15S);
			IF tonTimeOut.Q THEN
				_Abort := TRUE;
				uiResumeStep := uiExecutingStep;
				strStatus := M_FormatManagedStatus(
					AlarmId := GVL_ErrorCode.GC_ALARM_ALC_OUTROBOT_RARE,
					InnerMessage := GVL_ErrorCode.GC_MSG_0048);
				Status := strStatus;
				Error := TRUE;
			END_IF
		END_IF
	END_IF

1300: // Clip close (pick)
	IF bSyncPick THEN
		Clips[0].M_Extend();
		Clips[1].M_Extend();
		bCylinderCheck := Clips[0].InFrontPosition AND Clips[1].InFrontPosition;
	ELSE
		Clips[iWorkingIndex].M_Extend();
		bCylinderCheck := Clips[iWorkingIndex].InFrontPosition;
	END_IF
	IF bCylinderCheck THEN
		// Safety: 標記夾到箱 (sync 時兩爪都標)
		IF bSyncPick THEN
			bClipHasBox[0] := TRUE;
			bClipHasBox[1] := TRUE;
		ELSE
			bClipHasBox[iWorkingIndex] := TRUE;
		END_IF
		uiExecutingStep:=1400;
	ELSE
		tonTimeOut(IN:=TRUE, PT:=T#15S);
		IF tonTimeOut.Q THEN
			_Abort := TRUE;
			uiResumeStep := uiExecutingStep;
			strStatus := M_FormatManagedStatus(
				AlarmId := GVL_ErrorCode.GC_ALARM_ALC_OUTROBOT_RARE,
				InnerMessage := GVL_ErrorCode.GC_MSG_0026);
			Status := strStatus;
			Error := TRUE;
		END_IF
	END_IF

1400: // Clip up (pick) - 提箱離開 TT
	IF bSyncPick THEN
		Cylinders[0].M_Retract();
		Cylinders[1].M_Retract();
		bCylinderCheck := Cylinders[0].InRearPosition AND Cylinders[1].InRearPosition;
	ELSE
		Cylinders[iWorkingIndex].M_Retract();
		bCylinderCheck := Cylinders[iWorkingIndex].InRearPosition;
	END_IF
	IF bCylinderCheck THEN
		uiExecutingStep:=1500;
	ELSE
		tonTimeOut(IN:=TRUE, PT:=T#15S);
		IF tonTimeOut.Q THEN
			_Abort := TRUE;
			uiResumeStep := uiExecutingStep;
			strStatus := M_FormatManagedStatus(
				AlarmId := GVL_ErrorCode.GC_ALARM_ALC_OUTROBOT_RARE,
				InnerMessage := GVL_ErrorCode.GC_MSG_0050);
			Status := strStatus;
			Error := TRUE;
		END_IF
	END_IF

1500: // Next pick? (修雙 clip 漏放 bug, 用 bPickedA/B 旗標)
	IF bSyncPick THEN
		bPickedA := TRUE;
		bPickedB := TRUE;
	ELSIF iWorkingIndex = 0 THEN
		bPickedA := TRUE;
	ELSE
		bPickedB := TRUE;
	END_IF
	IF UseA AND NOT bPickedA THEN
		iWorkingIndex := 0;
		uiExecutingStep := 1000;
	ELSIF UseB AND NOT bPickedB THEN
		iWorkingIndex := 1;
		uiExecutingStep := 1000;
	ELSE
		// 全部 pick 完,進 1600 確認 R 上箱已離開
		IF UseA THEN
			iWorkingIndex := 0;
		ELSE
			iWorkingIndex := 1;
		END_IF
		uiExecutingStep := 1600;
	END_IF

1600: // Confirm box left R sensor (pick 真的有抓起來)
	IF (UseA AND INPUT.bTurnTable_R1Detect_Sensor) OR (UseB AND INPUT.bTurnTable_R2Detect_Sensor) THEN
		// 還偵測到箱 → 等 timeout 才報錯,因為氣缸抬起到感測器斷訊有延遲
		tonTimeOut(IN:=TRUE, PT:=T#15S);
		IF tonTimeOut.Q THEN
			_Abort := TRUE;
			uiResumeStep := uiExecutingStep;
			strStatus := M_FormatManagedStatus(
				AlarmId := GVL_ErrorCode.GC_ALARM_ALC_OUTROBOT_RARE,
				InnerMessage := GVL_ErrorCode.GC_MSG_0016);
		END_IF
	ELSE
		uiExecutingStep:=2000;
	END_IF

2000: // Move conveyor + send OutRobot to placing pos
	IF bMotorMoveForward THEN
		bMoveConveyorForward:=TRUE;
		bMoveConveyorBackrward:=FALSE;
	ELSE
		bMoveConveyorForward:=FALSE;
		bMoveConveyorBackrward:=TRUE;
	END_IF
	arAxisCtrl_gb[AxisNo.OutRobot_X].PosMode.Position := PlacingPos[iWorkingIndex].X_Pos;
	arAxisCtrl_gb[AxisNo.OutRobot_Y].PosMode.Position := PlacingPos[iWorkingIndex].Y_Pos;
	uiExecutingStep:=2100;

2100: // Wait OutRobot XY arrive + sensor 'no box at conveyor stop' for a while
	tonTimeDelay(IN:=NOT SensorOnConveyor, PT:=T#1S);
	IF (arAxisStatus_gb[AxisNo.OutRobot_X].Admin._OpModeAck = ModePosAbs AND arAxisStatus_gb[AxisNo.OutRobot_X].Admin.CmdDone)
	AND (arAxisStatus_gb[AxisNo.OutRobot_Y].Admin._OpModeAck = ModePosAbs AND arAxisStatus_gb[AxisNo.OutRobot_Y].Admin.CmdDone)
	AND tonTimeDelay.Q
	THEN
		uiExecutingStep:=2150;
	ELSE
		tonTimeOut(IN:=TRUE, PT:=T#15S);
		IF tonTimeOut.Q THEN
			_Abort := TRUE;
			uiResumeStep := 2000;
			strStatus := M_FormatManagedStatus(
				AlarmId := GVL_ErrorCode.GC_ALARM_ALC_OUTROBOT_RARE,
				InnerMessage := GVL_ErrorCode.GC_MSG_0129);
		END_IF
	END_IF

2150: // Stop conveyor
	bMoveConveyorForward := FALSE;
	bMoveConveyorBackrward := FALSE;
	ConveyorMotor.M_MotorStop();
	IF ConveyorMotor.InStopped THEN
		uiExecutingStep:=2200;
	END_IF
	

2200: // Clip down (place) - Fix 2: 下爪前位置再確認
	IF NOT M_IsOutRobotAtPos(TargetPos:=PlacingPos[iWorkingIndex]) THEN
		_Error := TRUE;
		uiResumeStep := uiExecutingStep;
		strStatus := M_FormatManagedStatus(
			AlarmId := GVL_ErrorCode.GC_ALARM_ALC_OUTROBOT_RARE,
			InnerMessage := GVL_ErrorCode.GC_MSG_0173);
		Status := strStatus;
		Error := TRUE;
	ELSE
		IF bSyncPlace THEN
			Cylinders[0].M_Extend();
			Cylinders[1].M_Extend();
			bCylinderCheck := Cylinders[0].InFrontPosition AND Cylinders[1].InFrontPosition;
		ELSE
			Cylinders[iWorkingIndex].M_Extend();
			bCylinderCheck := Cylinders[iWorkingIndex].InFrontPosition;
		END_IF
		IF bCylinderCheck THEN
			uiExecutingStep:=2300;
		ELSE
			tonTimeOut(IN:=TRUE, PT:=T#15S);
			IF tonTimeOut.Q THEN
				_Abort := TRUE;
				uiResumeStep := uiExecutingStep;
				strStatus := M_FormatManagedStatus(
					AlarmId := GVL_ErrorCode.GC_ALARM_ALC_OUTROBOT_RARE,
					InnerMessage := GVL_ErrorCode.GC_MSG_0051);
				Status := strStatus;
				Error := TRUE;
			END_IF
		END_IF
	END_IF

2300: // Clip open (place)
	IF bSyncPlace THEN
		Clips[0].M_Retract();
		Clips[1].M_Retract();
		bCylinderCheck := Clips[0].InRearPosition AND Clips[1].InRearPosition;
	ELSE
		Clips[iWorkingIndex].M_Retract();
		bCylinderCheck := Clips[iWorkingIndex].InRearPosition;
	END_IF
	IF bCylinderCheck THEN
		// Safety: 箱已放下 (sync 時兩爪都清)
		IF bSyncPlace THEN
			bClipHasBox[0] := FALSE;
			bClipHasBox[1] := FALSE;
		ELSE
			bClipHasBox[iWorkingIndex] := FALSE;
		END_IF
		uiExecutingStep:=2400;
	ELSE
		tonTimeOut(IN:=TRUE, PT:=T#15S);
		IF tonTimeOut.Q THEN
			_Abort := TRUE;
			uiResumeStep := uiExecutingStep;
			strStatus := M_FormatManagedStatus(
				AlarmId := GVL_ErrorCode.GC_ALARM_ALC_OUTROBOT_RARE,
				InnerMessage := GVL_ErrorCode.GC_MSG_0027);
			Status := strStatus;
			Error := TRUE;
		END_IF
	END_IF

2400: // Clip up (place)
	IF bSyncPlace THEN
		Cylinders[0].M_Retract();
		Cylinders[1].M_Retract();
		bCylinderCheck := Cylinders[0].InRearPosition AND Cylinders[1].InRearPosition;
	ELSE
		Cylinders[iWorkingIndex].M_Retract();
		bCylinderCheck := Cylinders[iWorkingIndex].InRearPosition;
	END_IF
	IF bCylinderCheck THEN
		uiExecutingStep:=2500;
	ELSE
		tonTimeOut(IN:=TRUE, PT:=T#15S);
		IF tonTimeOut.Q THEN
			_Abort := TRUE;
			uiResumeStep := uiExecutingStep;
			strStatus := M_FormatManagedStatus(
				AlarmId := GVL_ErrorCode.GC_ALARM_ALC_OUTROBOT_RARE,
				InnerMessage := GVL_ErrorCode.GC_MSG_0053);
			Status := strStatus;
			Error := TRUE;
		END_IF
	END_IF

2500: // Next place? (修雙 clip 漏放 bug, 用 bPlacedA/B 旗標)
	IF bSyncPlace THEN
		bPlacedA := TRUE;
		bPlacedB := TRUE;
	ELSIF iWorkingIndex = 0 THEN
		bPlacedA := TRUE;
	ELSE
		bPlacedB := TRUE;
	END_IF
	IF UseA AND NOT bPlacedA THEN
		iWorkingIndex := 0;
		uiExecutingStep := 2000;
	ELSIF UseB AND NOT bPlacedB THEN
		iWorkingIndex := 1;
		uiExecutingStep := 2000;
	ELSE
		uiExecutingStep := 2600;
	END_IF

2600: // Move conveyor a bit until box detected at conveyor stop
	IF bMotorMoveForward THEN
		bMoveConveyorForward:=TRUE;
	ELSE
		bMoveConveyorBackrward:=TRUE;
	END_IF
	tonTimeDelay(IN:=NOT SensorOnConveyor, PT:=T#1S);
	IF tonTimeDelay.Q THEN
		uiExecutingStep:=2700;
	ELSE
		tonTimeOut(IN:=TRUE, PT:=T#15S);
		IF tonTimeOut.Q THEN
			_Abort := TRUE;
			uiResumeStep := uiExecutingStep;
			strStatus := M_FormatManagedStatus(
				AlarmId := GVL_ErrorCode.GC_ALARM_ALC_OUTROBOT_RARE,
				InnerMessage := GVL_ErrorCode.GC_MSG_0081);
			Status := strStatus;
			Error := TRUE;
		END_IF
	END_IF

2700: // Stop motor
	bMoveConveyorForward:=FALSE;
	bMoveConveyorBackrward:=FALSE;
	ConveyorMotor.M_MotorStop();
	IF ConveyorMotor.InStopped THEN
		uiExecutingStep:=3000;
	END_IF

3000: // Finish
	bMoveConveyorForward:=FALSE;
	bMoveConveyorBackrward:=FALSE;
	_Executed:=TRUE;

END_CASE

IF NOT Execute THEN
	eState:=STATE_RESETTING;
END_IF
IF _Error THEN
	eState:=STATE_ERROR;
END_IF
IF _Abort THEN
	eSTATE:=STATE_ABORTING;
END_IF
IF _Executed THEN
	eSTATE:=STATE_Done;
END_IF
END_METHOD

METHOD  M_STATE_RESETTING
VAR_INPUT
END_VAR
Busy := TRUE;
Error := _Error;

// Timer 確保歸零
tonTimeOut(IN:=FALSE);
tonTimeDelay(IN:=FALSE);
tonLeaveDebounce(IN:=FALSE);

CASE uiResettingStep OF

	0:
		IF __ISVALIDREF(ConveyorMotor) THEN
			ConveyorMotor.M_MotorStop();
		END_IF
		M_RecoveryAllObjects();
		uiResettingStep:=9999;

	9999:
		Done := FALSE;
		Busy := FALSE;
		_ResetCompleted:=TRUE;
END_CASE
IF _ResetCompleted THEN
	eSTATE:=STATE_DORMANT;
END_IF
END_METHOD

END_FUNCTION_BLOCK

// ---- Library/20_MachineUnits/22_AllocateArea/Service/FB_OutRobot_BoxMoveReverse.TcPOU
FUNCTION_BLOCK FB_OutRobot_BoxMoveReverse EXTENDS FB_ObjectBase_V2
VAR_INPUT
//    Execute    :BOOL;   // True : This prog will start.
//    Abort      :BOOL;   // True : This prog will be abort.
//    Reset      :BOOL;   // True : This prog will be reset.
//    ObjectName :STRING; // Set this fb name(About it's action)
	INPUT            			   : REFERENCE TO ST_InputTable;
	Cylinder   					   : REFERENCE TO UNI_CylinderList;
	Motor      					   : REFERENCE TO UNI_MotorList;
	Cylinders					   : REFERENCE TO ARRAY[0..1] OF FB_Cylinder;
	Clips						   : REFERENCE TO ARRAY[0..1] OF FB_Cylinder;
	AutoMode_OutRobotMoveMove : st_AutoMode_ClampingBoxesJob;	
END_VAR

VAR_OUTPUT
//    Busy    :BOOL;        // True : This prog is running.
//    Done    :BOOL;        // True : Command has been executed.
//    Aborted :BOOL;        // True : This prog is aborted.
//    Error   :BOOL;        // True : This prog has an error.
//    ErrorID :UINT;       // Output ErrorID
//    Status  :T_MaxString; // Output this prog status by string(255bytes)
END_VAR

VAR
//    eState :E_MethodStatus_Basic;
//	uiExecutingStep : UDINT; // This var is used to been controll STATE_EXECUTING process.
//	uiResettingStep : UDINT;
//	uiAbortingStep : UDINT;
//	_Executed :BOOL; // Executing process completed.
//	_Error : BOOL; // FB has an error.
//	_ResetCompleted : BOOL; // FB resetting completed.
//	_AbortCompleted : BOOL; // FB aborting completed.
//	_Abort		: BOOL;
	strStatus	: STRING;
	uiResumeStep : UDINT;
	tonTimeOut   :TON;
	tonTimeDelay   :TON;
	iWorkingIndex : INT;
	_UniqueErrorCode :STRING;

	PickingPos	: ARRAY[0..1] OF ST_PositionTable;
	PlacingPos  : ARRAY[0..1] OF ST_PositionTable;
	bSyncPick	: BOOL;
	bSyncPlace	: BOOL;
	SensorOnConveyor			   : BIT;
	ConveyorMotor				   : REFERENCE TO FB_Motor;
	UseA	: BOOL;
	UseB	: BOOL;
	bMotorMoveForward : BOOL;
	lrEpsPos 	: LREAL := 0.001;	// 浮點座標比較容差 (sync 判斷)
	// Step 切換偵測 (timer 乾淨重置)
	uiExecutingStep_Last : UDINT;
	// Resume / Pause 機制
	bResumeEnabled : BOOL;
	bCanPause : BOOL;
	bPauseLast : BOOL;
	// 雙 clip pick / place 旗標 (取代 iWorkingIndex 共用)
	bPickedA : BOOL;
	bPickedB : BOOL;
	bPlacedA : BOOL;
	bPlacedB : BOOL;
	// Safety: 夾爪是否正夾著箱 (latched, 1300 閉夾→TRUE, 2300 開夾→FALSE)
	bClipHasBox : ARRAY[0..1] OF BOOL;
	
	_bRetry  : BOOL;
	
	// Error blinking 閃爍邏輯
	trigErrorReset		: R_TRIG;
	tonErrorResetDelay	: TON;
	bErrorBlinking		: BOOL;
END_VAR

A00_BasicUnits();
SUPER^.A10_StateControl();

ACTION A00_BasicUnits:
// Timer 由各 step 自行呼叫並傳 IN/PT,此處不做 freerun call,
// 避免「IN 殘留 TRUE」造成 step 切換後 timer 不歸零。
END_ACTION

METHOD GetModelState
VAR_OUTPUT
    xDone    :BOOL;
    xBusy    :BOOL;
    xError   :BOOL;
    xAborted :BOOL;
    iErrorID :UDINT;
	UniqueErrorCode : STRING;
END_VAR
xDone    := Done;
xBusy    := Busy;
xError   := Error;
xAborted := Aborted;
iErrorID := ErrorID;
UniqueErrorCode := THIS^.UniqueErrorCode;
END_METHOD

METHOD GetName : STRING
GetName := ObjectName;
END_METHOD

METHOD PRIVATE M_CheckCommand : BOOL
VAR_INPUT
END_VAR
IF NOT AutoMode_OutRobotMoveMove.ClampingInfo.UseClibA AND NOT AutoMode_OutRobotMoveMove.ClampingInfo.UseClibB THEN
	M_CheckCommand := FALSE;
	strStatus 	   := 'FB_OutRobot_BoxMoveReverse , Wrong Command Neither Clamp was used';
	RETURN;
END_IF
IF AutoMode_OutRobotMoveMove.ClampingInfo.TargetOfClipA <> AutoMode_OutRobotMoveMove.ClampingInfo.TargetOfClipB THEN
	M_CheckCommand := FALSE;
	strStatus 	   := 'FB_OutRobot_BoxMoveReverse , Wrong Command ClampA,B need same TargetPos';
	RETURN;
END_IF

M_CheckCommand:=true;
END_METHOD

METHOD PRIVATE M_GetResumeEntryStep : UDINT
VAR_INPUT
	uiErrorStep : UDINT;
END_VAR
// Resume 入口對照表: 錯誤點 → 重新進入的安全 checkpoint
CASE uiErrorStep OF
	1000, 1100:
		M_GetResumeEntryStep := 1000;
	1200, 1300, 1400, 1500, 1600:
		M_GetResumeEntryStep := 1000;	// pick 階段錯誤 → 重發 XY 從頭 pick
	2000, 2100, 2150:
		M_GetResumeEntryStep := 2000;
	2200, 2300, 2400, 2500:
		M_GetResumeEntryStep := 2000;	// place 階段錯誤 → 重發 XY 從頭 place
	2600, 2700:
		M_GetResumeEntryStep := 2600;	// conveyor handoff 重做
ELSE
	M_GetResumeEntryStep := 0;
END_CASE
END_METHOD

METHOD PRIVATE M_GetWorkingConditions : BOOL
VAR_INPUT
END_VAR
//For Outbox move reverse, Boxes must place on same position , therefor only work with TargetPosition of ClipA



IF AutoMode_OutRobotMoveMove.ClampingInfo.TargetOfClipA = 5 THEN
	ConveyorMotor REF= Motor.List.TransmitDifferentSideCV;
ELSIF AutoMode_OutRobotMoveMove.ClampingInfo.TargetOfClipA = 6 THEN
	ConveyorMotor REF= Motor.List.TransmitSameSideCV;
ELSIF AutoMode_OutRobotMoveMove.ClampingInfo.TargetOfClipA = 3 THEN
	ConveyorMotor REF= Motor.List.TransmitDifferentSideCV;
ELSIF AutoMode_OutRobotMoveMove.ClampingInfo.TargetOfClipA = 4 THEN
	ConveyorMotor REF= Motor.List.TransmitSameSideCV;
END_IF

IF AutoMode_OutRobotMoveMove.ClampingInfo.TargetOfClipA=5 THEN
		bMotorMoveForward := FALSE;
	ELSE
		bMotorMoveForward := TRUE;
END_IF
IF AutoMode_OutRobotMoveMove.ClampingInfo.UseClibA THEN
	PickingPos[0] :=FUN_GetPositionTableData('R',1,0);
	UseA := TRUE;
	CASE  AutoMode_OutRobotMoveMove.ClampingInfo.TargetOfClipA OF

	3,4:
		PlacingPos[0] :=FUN_GetPositionTableData('O',AutoMode_OutRobotMoveMove.ClampingInfo.TargetOfClipA,0);
	5,6:
		PlacingPos[0] :=FUN_GetPositionTableData('I',AutoMode_OutRobotMoveMove.ClampingInfo.TargetOfClipA,0);
	ELSE
		strStatus := M_FormatManagedStatus(
			AlarmId := GVL_ErrorCode.GC_ALARM_ALC_OUTROBOT_REVERSE,
			InnerMessage := GVL_ErrorCode.GC_MSG_0157);
		Status := strStatus;
		Error := TRUE;
		M_GetWorkingConditions := FALSE;
		RETURN;
	END_CASE
END_IF

IF AutoMode_OutRobotMoveMove.ClampingInfo.UseClibB THEN
	PickingPos[1] :=FUN_GetPositionTableData('R',2,1);
	UseB :=TRUE;
		CASE AutoMode_OutRobotMoveMove.ClampingInfo.TargetOfClipB OF

	3,4:
		PlacingPos[1] :=FUN_GetPositionTableData('O',AutoMode_OutRobotMoveMove.ClampingInfo.TargetOfClipB,1);
	5,6 :
		PlacingPos[1] :=FUN_GetPositionTableData('I',AutoMode_OutRobotMoveMove.ClampingInfo.TargetOfClipB,1);
	ELSE
		strStatus := M_FormatManagedStatus(
			AlarmId := GVL_ErrorCode.GC_ALARM_ALC_OUTROBOT_REVERSE,
			InnerMessage := GVL_ErrorCode.GC_MSG_0158);
		Status := strStatus;
		Error := TRUE;
		M_GetWorkingConditions := FALSE;
		RETURN;
	END_CASE
END_IF

// Sync 判斷一律用浮點容差 (lrEpsPos), OutRobot 只有 X/Y 軸 (無 R 軸),
// 不比較 R_Pos 避免因不相關欄位微誤差導致 sync 永遠 FALSE
bSyncPlace := UseA AND UseB
	AND ABS(PlacingPos[0].X_Pos - PlacingPos[1].X_Pos) < lrEpsPos
	AND ABS(PlacingPos[0].Y_Pos - PlacingPos[1].Y_Pos) < lrEpsPos;

bSyncPick := UseA AND UseB
	AND ABS(PickingPos[0].X_Pos - PickingPos[1].X_Pos) < lrEpsPos
	AND ABS(PickingPos[0].Y_Pos - PickingPos[1].Y_Pos) < lrEpsPos;

M_GetWorkingConditions :=TRUE;
END_METHOD

METHOD PRIVATE M_IsOutRobotAtPos : BOOL
VAR_INPUT
	TargetPos : ST_PositionTable;
END_VAR
VAR
	lTol : LREAL := 0.1;
END_VAR
//lTol := GVL_HMI.Setup.Mechanical.OutRobotPositionTolerance;

M_IsOutRobotAtPos :=
		NOT arAxisCtrl_gb[AxisNo.OutRobot_X].Admin.Axis.Status.Moving
	AND NOT arAxisCtrl_gb[AxisNo.OutRobot_Y].Admin.Axis.Status.Moving
	AND ABS(arAxisCtrl_gb[AxisNo.OutRobot_X].Admin.Axis.NcToPlc.ActPos - TargetPos.X_Pos) < lTol
	AND ABS(arAxisCtrl_gb[AxisNo.OutRobot_Y].Admin.Axis.NcToPlc.ActPos - TargetPos.Y_Pos) < lTol;
END_METHOD

METHOD PRIVATE M_IsTurnTableAtStation : BOOL
VAR
	lActPos : LREAL;
	lTol    : LREAL := 0.1;
END_VAR
// Pick 前 TurnTable 必須位於 0/90/180/270/360 (任一 station)
// 取絕對值處理負角度 (e.g., -90 → 90, -180 → 180)
lActPos := ABS(arAxisCtrl_gb[AxisNo.TurnTable].Admin.Axis.NcToPlc.ModuloActPos);

M_IsTurnTableAtStation :=
	   FUN_CheckInPos(ActPos:=lActPos, TargetPos:=0,   ToleranceRange:=lTol)
	OR FUN_CheckInPos(ActPos:=lActPos, TargetPos:=90,  ToleranceRange:=lTol)
	OR FUN_CheckInPos(ActPos:=lActPos, TargetPos:=180, ToleranceRange:=lTol)
	OR FUN_CheckInPos(ActPos:=lActPos, TargetPos:=270, ToleranceRange:=lTol)
	OR FUN_CheckInPos(ActPos:=lActPos, TargetPos:=360, ToleranceRange:=lTol);
END_METHOD

METHOD PRIVATE M_RecoveryAllObjects : BOOL
VAR_INPUT
END_VAR
VAR 
	i : INT;
END_VAR
FOR i:=0 TO 1 DO
	// Clip: 有箱時絕對不張開 (safety),只清錯
	IF Clips[i].xError THEN
		Clips[i].M_Reset();
	ELSIF NOT bClipHasBox[i] THEN
		Clips[i].M_Retract();
	END_IF
	// Cylinder: 一律抬起 (空爪或有箱都安全)
	IF Cylinders[i].xError THEN
		Cylinders[i].M_Reset();
	ELSE
		Cylinders[i].M_Retract();
	END_IF
END_FOR


IF arAxisCtrl_gb[AxisNo.OutRobot_X].Admin.Axis.Status.Error THEN

	arAxisCtrl_gb[AxisNo.OutRobot_X].Admin.ClearError:= TRUE;
ELSE
	arAxisCtrl_gb[AxisNo.OutRobot_X].Admin.ClearError:= FALSE;
END_IF

IF arAxisCtrl_gb[AxisNo.OutRobot_Y].Admin.Axis.Status.Error THEN

	arAxisCtrl_gb[AxisNo.OutRobot_Y].Admin.ClearError:= TRUE;
ELSE
	arAxisCtrl_gb[AxisNo.OutRobot_Y].Admin.ClearError:= FALSE;
END_IF
END_METHOD

METHOD PRIVATE M_SensorUpdate : BOOL
VAR_INPUT
END_VAR
IF AutoMode_OutRobotMoveMove.ClampingInfo.TargetOfClipA = 5 THEN
	SensorOnConveyor := INPUT.bDifferentSizeCV_BoxDetect5_Sensor;
ELSIF AutoMode_OutRobotMoveMove.ClampingInfo.TargetOfClipA = 6 THEN
	SensorOnConveyor := INPUT.bSameSizeCV_BoxDetect5_Sensor;
ELSIF AutoMode_OutRobotMoveMove.ClampingInfo.TargetOfClipA = 3 THEN
	SensorOnConveyor := INPUT.bDifferentSizeCV_BoxDetect4_Sensor;
ELSIF AutoMode_OutRobotMoveMove.ClampingInfo.TargetOfClipA = 4 THEN
	SensorOnConveyor := INPUT.bSameSizeCV_BoxDetect4_Sensor;	
END_IF
END_METHOD

METHOD  M_STATE_ABORTED
VAR_INPUT
END_VAR
IF NOT _bRetry THEN
	ERROR 			:= TRUE;
	Busy    		:= FALSE;
	Aborted 		:= TRUE;
	Status 			:= strStatus;
	uiAbortingStep  := 0;
	_AbortCompleted := TRUE;
END_IF

IF reset THEN
	ERROR 	:= FALSE;
	Aborted := FALSE;
	_bRetry	:= TRUE;
END_IF

IF NOT Execute THEN
	eSTATE:=STATE_RESETTING;
// 續做: Reset+Execute 時設旗標,EXECUTING step 0 會跳到 ResumeStep
ELSIF Execute AND _bRetry AND uiResumeStep > 0 THEN
	Status  := '';
	bResumeEnabled := TRUE;
	uiExecutingStep := 0;
	eSTATE:=STATE_EXECUTING;
// 判斷如果是不能續做的，重新跳回aborting 再次進入aborted 循環，上位下Reset 會看Error 如果Error沒有消失會卡住。
ELSIF Execute AND _bRetry AND uiResumeStep = 0 THEN	
	strStatus := 'FB_OutRobot_BoxMoveReverse, this Error can not retry';
	eState := STATE_ERROR;
END_IF
END_METHOD

METHOD  M_STATE_ABORTING
VAR_INPUT
END_VAR

VAR
	i : int;
	bCylinderCheck: BOOL;
END_VAR
// Timer 歸零
tonTimeOut(IN:=FALSE);
tonTimeDelay(IN:=FALSE);

CASE uiAbortingStep OF
	0 :
		_Abort  := FALSE;
		_bRetry := FALSE;
		bCylinderCheck:=TRUE;
		IF __ISVALIDREF(ConveyorMotor) THEN
			ConveyorMotor.M_MotorStop();
		END_IF

		// Safety: 有箱的 clip 絕對不張開
		FOR i :=0 TO 1 DO
			IF Clips[i].xError THEN
				Clips[i].M_Reset();
			ELSIF NOT bClipHasBox[i] THEN
				Clips[i].M_Retract();
			END_IF
		END_FOR

		// Cylinder 一律抬起 (空爪或有箱都安全)
		FOR i :=0 TO 1 DO
			IF Cylinders[i].xError THEN
				Cylinders[i].M_Reset();
			END_IF
			Cylinders[i].M_Retract();
			bCylinderCheck:=bCylinderCheck AND Cylinders[i].InRearPosition;
		END_FOR

		IF bCylinderCheck THEN
			uiAbortingStep:=9999;
		END_IF

	9999:
		_Abort := FALSE;
		_AbortCompleted:=TRUE;
END_CASE

IF NOT Execute THEN
	eState := STATE_RESETTING;
ELSIF Execute AND _AbortCompleted THEN
	eSTATE :=STATE_ABORTED;
END_IF
END_METHOD

METHOD  M_STATE_DONE
VAR_INPUT
END_VAR
Busy 	:= FALSE;
Done	:=TRUE;

IF NOT Execute THEN
	eSTATE:=STATE_RESETTING;
END_IF
END_METHOD

METHOD  M_STATE_DORMANT
VAR_INPUT
END_VAR
Busy            := FALSE;
Done            := FALSE;
Aborted         := FALSE;
Error           := FALSE;
ErrorID         := 0;
Status          := '';
_ResetCompleted := FALSE;
_Error          := FALSE;
_Executed       := FALSE;
_Abort          := FALSE;
strStatus := M_FormatManagedStatus(
	AlarmId := GVL_ErrorCode.GC_ALARM_ALC_OUTROBOT_REVERSE,
	InnerMessage := GVL_ErrorCode.GC_MSG_0089);
Status := '';
Error := FALSE;
uiExecutingStep :=uiResettingStep :=0;
// Timer 完整歸零 (用實際 FB call,不是只設屬性)
tonTimeOut(IN:=FALSE);
tonTimeDelay(IN:=FALSE);
uiExecutingStep_Last := 0;
_UniqueErrorCode:='0';
iWorkingIndex :=0;
bSyncPick := FALSE;
bSyncPlace := FALSE;
UseA := FALSE;
UseB := FALSE;
bMotorMoveForward := FALSE;
bPickedA := FALSE;
bPickedB := FALSE;
bPlacedA := FALSE;
bPlacedB := FALSE;
bPauseLast 	:= FALSE;
bCanPause 	:= FALSE;
_bRetry	 	:= FALSE;
_AbortCompleted := FALSE;
uiAbortingStep  := 0;
tonErrorResetDelay.IN := FALSE;
// 非續做模式才清 ResumeStep 與 ClipHasBox
IF NOT bResumeEnabled THEN
	uiResumeStep := 0;
	bClipHasBox[0] := FALSE;
	bClipHasBox[1] := FALSE;
END_IF
// 註: M_RecoveryAllObjects 不放 DORMANT 避免與其他 FB 搶 ClearError,
// 以及避免清掉 bClipHasBox 後誤張爪掉箱。僅 EXECUTING step 0 / RESETTING 呼叫。

IF Execute THEN
	eSTATE:=STATE_EXECUTING;
END_IF
END_METHOD

METHOD  M_STATE_ERROR
VAR_INPUT
END_VAR
ERROR   :=TRUE;
Busy	:=FALSE;
_Error  := FALSE;
Status := strStatus;
IF __ISVALIDREF(ConveyorMotor) THEN
	ConveyorMotor.M_MotorStop();
END_IF

// --- Reset 閃爍邏輯：偵測上升緣觸發 1 秒閃爍 ---
trigErrorReset(CLK := reset);
IF trigErrorReset.Q THEN
	bErrorBlinking := TRUE;
END_IF

tonErrorResetDelay(IN := bErrorBlinking, PT := T#1S);
IF tonErrorResetDelay.Q THEN
	bErrorBlinking := FALSE;
END_IF

// 閃爍期間 (1秒) 暫時將 Error 訊號設為 FALSE
IF bErrorBlinking THEN
	Error := FALSE;
END_IF


IF NOT Execute THEN
	bErrorBlinking := FALSE;
	tonErrorResetDelay.IN := FALSE;
	eSTATE:=STATE_RESETTING;
END_IF
END_METHOD

METHOD  M_STATE_EXECUTING
VAR_INPUT
END_VAR
VAR_INST
	bMoveConveyorForward : BOOL;
	bMoveConveyorBackrward : bool;
END_VAR

VAR
	bCylinderCheck : BOOL := TRUE;
END_VAR
Busy :=TRUE;
M_SensorUpdate();

// ============================================================
// (A) Step 切換 → Timer 完整歸零 (Fix 1)
// ============================================================
IF uiExecutingStep <> uiExecutingStep_Last THEN
	tonTimeOut(IN:=FALSE);
	tonTimeDelay(IN:=FALSE);
	uiExecutingStep_Last := uiExecutingStep;
END_IF

// ============================================================
// (B) TurnTable Interlock (Fix 3)
// Pick 下爪區間 (1200~1499) 期間 TurnTable 不可移動
// ============================================================
IF (uiExecutingStep >= 1200 AND uiExecutingStep <= 1499) THEN
	IF arAxisCtrl_gb[AxisNo.TurnTable].Admin.Axis.Status.Moving THEN
		_Error := TRUE;
		uiResumeStep := uiExecutingStep;
		strStatus := M_FormatManagedStatus(
			AlarmId := GVL_ErrorCode.GC_ALARM_ALC_OUTROBOT_REVERSE,
			InnerMessage := GVL_ErrorCode.GC_MSG_0174);
		Status := strStatus;
		Error := TRUE;
	END_IF
END_IF

// ============================================================
// (C) Pause 處理 (Fix 4) - 僅在「安全 step」生效
// ============================================================
bCanPause :=
	   uiExecutingStep = 0
	OR uiExecutingStep = 100
	OR uiExecutingStep = 200
	OR uiExecutingStep = 1000
	OR uiExecutingStep = 1100
	OR uiExecutingStep = 1500
	OR uiExecutingStep = 2000
	OR uiExecutingStep = 2100
	OR uiExecutingStep = 2150
	OR uiExecutingStep = 2500
	OR uiExecutingStep = 2700;

// Pause 釋放邊緣 → 強制 timer 歸零
IF bPauseLast AND NOT Pause THEN
	tonTimeOut(IN:=FALSE);
	tonTimeDelay(IN:=FALSE);
END_IF
bPauseLast := Pause;

IF Pause AND bCanPause THEN
	bMoveConveyorForward := FALSE;
	bMoveConveyorBackrward := FALSE;
	IF __ISVALIDREF(ConveyorMotor) THEN
		ConveyorMotor.M_MotorStop();
	END_IF
	tonTimeOut(IN:=FALSE);
	tonTimeDelay(IN:=FALSE);
	Busy := TRUE;
	RETURN;
END_IF

// ============================================================
// Conveyor 連續控制 (sync 後 latched flag 控制)
// ============================================================
IF bMoveConveyorForward THEN
	IF NOT ConveyorMotor.InBackWard THEN
		ConveyorMotor.M_MoveForward();
	END_IF
END_IF

IF bMoveConveyorBackrward THEN
	IF NOT ConveyorMotor.InForWard THEN
		ConveyorMotor.M_MoveBackward();
	END_IF
END_IF

CASE uiExecutingStep OF

0: //Entry - VAR_INST reset + 流程分流
	// VAR_INST 私有給本 method,DORMANT 看不到,必須在此 reset
	bMoveConveyorForward := FALSE;
	bMoveConveyorBackrward := FALSE;

	IF GVL_Machine.PackTags[UnitNo.Allocate].Status.UnitModeCurrent <> E_UnitMode.Auto THEN
		strStatus := 'Not in Auto mode';
		_UniqueErrorCode := 'E_NOT_AUTO_MODE';
		_Error := TRUE;
	ELSIF bResumeEnabled AND uiResumeStep > 0 THEN
		// 續做模式
		IF M_GetWorkingConditions() THEN
			M_RecoveryAllObjects();
			// Safety: 若仍夾著箱,強制走 placing 流程
			IF bClipHasBox[0] OR bClipHasBox[1] THEN
				IF bClipHasBox[0] THEN
					iWorkingIndex := 0;
				ELSE
					iWorkingIndex := 1;
				END_IF
				bPickedA := UseA;
				bPickedB := UseB;
				bPlacedA := UseA AND NOT bClipHasBox[0];
				bPlacedB := UseB AND NOT bClipHasBox[1];
				uiExecutingStep := 2000;
			ELSE
				uiExecutingStep := M_GetResumeEntryStep(uiErrorStep:=uiResumeStep);
			END_IF
			bResumeEnabled := FALSE;
			uiResumeStep := 0;
		ELSE
			_Error := TRUE;
		END_IF
	ELSE
		// 正常啟動: DORMANT 已 reset 所有 FB-level flag
		IF M_GetWorkingConditions() THEN
			M_RecoveryAllObjects();
			uiExecutingStep := 100;
		ELSE
			_Error := TRUE;
		END_IF
	END_IF

100: //Check command
	IF M_CheckCommand() THEN
		uiExecutingStep:=200;
	ELSE
		_Error :=TRUE;
	END_IF

200: // TT angle gate + 確認 R 上有箱
	IF NOT M_IsTurnTableAtStation() THEN
		_Abort := TRUE;
		uiResumeStep := uiExecutingStep;
		strStatus := M_FormatManagedStatus(
			AlarmId := GVL_ErrorCode.GC_ALARM_ALC_OUTROBOT_REVERSE,
			InnerMessage := GVL_ErrorCode.GC_MSG_0175);
	ELSIF (UseA AND NOT INPUT.bTurnTable_R1Detect_Sensor) OR (UseB AND NOT INPUT.bTurnTable_R2Detect_Sensor) THEN
		_Error:=TRUE;
		uiResumeStep := 0;	// 沒箱可抓 → 不可續做
		strStatus := M_FormatManagedStatus(
			AlarmId := GVL_ErrorCode.GC_ALARM_ALC_OUTROBOT_REVERSE,
			InnerMessage := GVL_ErrorCode.GC_MSG_0009);
		Status := strStatus;
		Error := TRUE;
	ELSE
		IF UseA THEN
			iWorkingIndex :=0;
		ELSE
			iWorkingIndex :=1;
		END_IF
		uiExecutingStep:=1000;
	END_IF

1000: // Move OutRobot to picking pos (TurnTable R)
	arAxisCtrl_gb[AxisNo.OutRobot_X].PosMode.Position := PickingPos[iWorkingIndex].X_Pos;
	arAxisCtrl_gb[AxisNo.OutRobot_Y].PosMode.Position := PickingPos[iWorkingIndex].Y_Pos;
	uiExecutingStep:=1100;

1100: // Wait OutRobot XY arrive (pick on TT) - 修正: 等 TurnTable 靜止 (原本誤檢查 RoundBelt)
	IF (arAxisStatus_gb[AxisNo.OutRobot_X].Admin._OpModeAck = ModePosAbs AND arAxisStatus_gb[AxisNo.OutRobot_X].Admin.CmdDone)
	AND (arAxisStatus_gb[AxisNo.OutRobot_Y].Admin._OpModeAck = ModePosAbs AND arAxisStatus_gb[AxisNo.OutRobot_Y].Admin.CmdDone)
	AND NOT arAxisCtrl_gb[AxisNo.TurnTable].Admin.Axis.Status.Moving
	THEN
		uiExecutingStep:=1200;
	ELSE
		tonTimeOut(IN:=TRUE, PT:=T#15S);
		IF tonTimeOut.Q THEN
			_Abort := TRUE;
			uiResumeStep := uiExecutingStep;
			strStatus := M_FormatManagedStatus(
				AlarmId := GVL_ErrorCode.GC_ALARM_ALC_OUTROBOT_REVERSE,
				InnerMessage := GVL_ErrorCode.GC_MSG_0082);
		END_IF
	END_IF

1200: // Clip down (pick) - Fix 2: 下爪前位置再確認
	IF NOT M_IsOutRobotAtPos(TargetPos:=PickingPos[iWorkingIndex]) THEN
		_Abort := TRUE;
		uiResumeStep := uiExecutingStep;
		strStatus := M_FormatManagedStatus(
			AlarmId := GVL_ErrorCode.GC_ALARM_ALC_OUTROBOT_REVERSE,
			InnerMessage := GVL_ErrorCode.GC_MSG_0172);
	ELSE
		// Sync 對稱化: sync 時兩爪同動同檢查
		IF bSyncPick THEN
			Cylinders[0].M_Extend();
			Cylinders[1].M_Extend();
			bCylinderCheck := Cylinders[0].InFrontPosition AND Cylinders[1].InFrontPosition;
		ELSE
			Cylinders[iWorkingIndex].M_Extend();
			bCylinderCheck := Cylinders[iWorkingIndex].InFrontPosition;
		END_IF
		IF bCylinderCheck THEN
			uiExecutingStep:=1300;
		ELSE
			tonTimeOut(IN:=TRUE, PT:=T#15S);
			IF tonTimeOut.Q THEN
				_Abort := TRUE;
				uiResumeStep := uiExecutingStep;
				strStatus := M_FormatManagedStatus(
					AlarmId := GVL_ErrorCode.GC_ALARM_ALC_OUTROBOT_REVERSE,
					InnerMessage := GVL_ErrorCode.GC_MSG_0048);
				Status := strStatus;
				Error := TRUE;
			END_IF
		END_IF
	END_IF

1300: // Clip close (pick)
	IF bSyncPick THEN
		Clips[0].M_Extend();
		Clips[1].M_Extend();
		bCylinderCheck := Clips[0].InFrontPosition AND Clips[1].InFrontPosition;
	ELSE
		Clips[iWorkingIndex].M_Extend();
		bCylinderCheck := Clips[iWorkingIndex].InFrontPosition;
	END_IF
	IF bCylinderCheck THEN
		// Safety: 標記夾到箱
		IF bSyncPick THEN
			bClipHasBox[0] := TRUE;
			bClipHasBox[1] := TRUE;
		ELSE
			bClipHasBox[iWorkingIndex] := TRUE;
		END_IF
		uiExecutingStep:=1400;
	ELSE
		tonTimeOut(IN:=TRUE, PT:=T#15S);
		IF tonTimeOut.Q THEN
			_Abort := TRUE;
			uiResumeStep := uiExecutingStep;
			strStatus := M_FormatManagedStatus(
				AlarmId := GVL_ErrorCode.GC_ALARM_ALC_OUTROBOT_REVERSE,
				InnerMessage := GVL_ErrorCode.GC_MSG_0025);
			Status := strStatus;
			Error := TRUE;
		END_IF
	END_IF

1400: // Clip up (pick)
	IF bSyncPick THEN
		Cylinders[0].M_Retract();
		Cylinders[1].M_Retract();
		bCylinderCheck := Cylinders[0].InRearPosition AND Cylinders[1].InRearPosition;
	ELSE
		Cylinders[iWorkingIndex].M_Retract();
		bCylinderCheck := Cylinders[iWorkingIndex].InRearPosition;
	END_IF
	IF bCylinderCheck THEN
		uiExecutingStep:=1500;
	ELSE
		tonTimeOut(IN:=TRUE, PT:=T#15S);
		IF tonTimeOut.Q THEN
			_Abort := TRUE;
			uiResumeStep := uiExecutingStep;
			strStatus := M_FormatManagedStatus(
				AlarmId := GVL_ErrorCode.GC_ALARM_ALC_OUTROBOT_REVERSE,
				InnerMessage := GVL_ErrorCode.GC_MSG_0049);
			Status := strStatus;
			Error := TRUE;
		END_IF
	END_IF

1500: // Next pick? (修雙 clip 漏放 bug, 用 bPickedA/B 旗標)
	IF bSyncPick THEN
		bPickedA := TRUE;
		bPickedB := TRUE;
	ELSIF iWorkingIndex = 0 THEN
		bPickedA := TRUE;
	ELSE
		bPickedB := TRUE;
	END_IF
	IF UseA AND NOT bPickedA THEN
		iWorkingIndex := 0;
		uiExecutingStep := 1000;
	ELSIF UseB AND NOT bPickedB THEN
		iWorkingIndex := 1;
		uiExecutingStep := 1000;
	ELSE
		// 全部 pick 完,先確認 R 上箱已離開,再進 placing
		IF UseA THEN
			iWorkingIndex := 0;
		ELSE
			iWorkingIndex := 1;
		END_IF
		uiExecutingStep := 1600;
	END_IF

1600: // Confirm box left R sensor (pick 真的有抓起來)
	IF (UseA AND INPUT.bTurnTable_R1Detect_Sensor) OR (UseB AND INPUT.bTurnTable_R2Detect_Sensor) THEN
		// 還偵測到箱 → 等 timeout 才報錯,因為氣缸抬起到感測器斷訊可能有延遲
		tonTimeOut(IN:=TRUE, PT:=T#15S);
		IF tonTimeOut.Q THEN
			_Abort := TRUE;
			uiResumeStep := uiExecutingStep;
			strStatus := M_FormatManagedStatus(
				AlarmId := GVL_ErrorCode.GC_ALARM_ALC_OUTROBOT_REVERSE,
				InnerMessage := GVL_ErrorCode.GC_MSG_0016);
			Status := strStatus;
			Error := TRUE;
		END_IF
	ELSE
		uiExecutingStep := 2000;
	END_IF


2000: // Move conveyor + send OutRobot to placing pos
	IF bMotorMoveForward THEN
		bMoveConveyorForward:=TRUE;
		bMoveConveyorBackrward:=FALSE;
	ELSE
		bMoveConveyorForward:=FALSE;
		bMoveConveyorBackrward:=TRUE;
	END_IF
	arAxisCtrl_gb[AxisNo.OutRobot_X].PosMode.Position := PlacingPos[iWorkingIndex].X_Pos;
	arAxisCtrl_gb[AxisNo.OutRobot_Y].PosMode.Position := PlacingPos[iWorkingIndex].Y_Pos;
	uiExecutingStep:=2100;

2100: // Wait OutRobot XY arrive + sensor 'no box at conveyor stop' for a while
	tonTimeDelay(IN:=NOT SensorOnConveyor, PT:=T#1S);
	IF (arAxisStatus_gb[AxisNo.OutRobot_X].Admin._OpModeAck = ModePosAbs AND arAxisStatus_gb[AxisNo.OutRobot_X].Admin.CmdDone)
	AND (arAxisStatus_gb[AxisNo.OutRobot_Y].Admin._OpModeAck = ModePosAbs AND arAxisStatus_gb[AxisNo.OutRobot_Y].Admin.CmdDone)
	AND tonTimeDelay.Q
	THEN
		uiExecutingStep:=2150;
	ELSE
		tonTimeOut(IN:=TRUE, PT:=T#15S);
		IF tonTimeOut.Q THEN
			_Abort := TRUE;
			uiResumeStep := uiExecutingStep;
			strStatus := M_FormatManagedStatus(
				AlarmId := GVL_ErrorCode.GC_ALARM_ALC_OUTROBOT_REVERSE,
				InnerMessage := GVL_ErrorCode.GC_MSG_0085);
		END_IF
	END_IF

2150: // Stop conveyor
	bMoveConveyorForward := FALSE;
	bMoveConveyorBackrward := FALSE;
	ConveyorMotor.M_MotorStop();
	IF ConveyorMotor.InStopped THEN
		uiExecutingStep:=2200;
	END_IF

2200: // Clip down (place) - Fix 2: 下爪前位置再確認
	IF NOT M_IsOutRobotAtPos(TargetPos:=PlacingPos[iWorkingIndex]) THEN
		_Abort := TRUE;
		uiResumeStep := uiExecutingStep;
		strStatus := M_FormatManagedStatus(
			AlarmId := GVL_ErrorCode.GC_ALARM_ALC_OUTROBOT_REVERSE,
			InnerMessage := GVL_ErrorCode.GC_MSG_0173);
	ELSE
		IF bSyncPlace THEN
			Cylinders[0].M_Extend();
			Cylinders[1].M_Extend();
			bCylinderCheck := Cylinders[0].InFrontPosition AND Cylinders[1].InFrontPosition;
		ELSE
			Cylinders[iWorkingIndex].M_Extend();
			bCylinderCheck := Cylinders[iWorkingIndex].InFrontPosition;
		END_IF
		IF bCylinderCheck THEN
			uiExecutingStep:=2300;
		ELSE
			tonTimeOut(IN:=TRUE, PT:=T#15S);
			IF tonTimeOut.Q THEN
				_Abort := TRUE;
				uiResumeStep := uiExecutingStep;
				strStatus := M_FormatManagedStatus(
					AlarmId := GVL_ErrorCode.GC_ALARM_ALC_OUTROBOT_REVERSE,
					InnerMessage := GVL_ErrorCode.GC_MSG_0051);
			END_IF
		END_IF
	END_IF

2300: // Clip open (place)
	IF bSyncPlace THEN
		Clips[0].M_Retract();
		Clips[1].M_Retract();
		bCylinderCheck := Clips[0].InRearPosition AND Clips[1].InRearPosition;
	ELSE
		Clips[iWorkingIndex].M_Retract();
		bCylinderCheck := Clips[iWorkingIndex].InRearPosition;
	END_IF
	IF bCylinderCheck THEN
		// Safety: 箱已放下
		IF bSyncPlace THEN
			bClipHasBox[0] := FALSE;
			bClipHasBox[1] := FALSE;
		ELSE
			bClipHasBox[iWorkingIndex] := FALSE;
		END_IF
		uiExecutingStep:=2400;
	ELSE
		tonTimeOut(IN:=TRUE, PT:=T#15S);
		IF tonTimeOut.Q THEN
			_Abort := TRUE;
			uiResumeStep := uiExecutingStep;
			strStatus := M_FormatManagedStatus(
				AlarmId := GVL_ErrorCode.GC_ALARM_ALC_OUTROBOT_REVERSE,
				InnerMessage := GVL_ErrorCode.GC_MSG_0028);
		END_IF
	END_IF

2400: // Clip up (place)
	IF bSyncPlace THEN
		Cylinders[0].M_Retract();
		Cylinders[1].M_Retract();
		bCylinderCheck := Cylinders[0].InRearPosition AND Cylinders[1].InRearPosition;
	ELSE
		Cylinders[iWorkingIndex].M_Retract();
		bCylinderCheck := Cylinders[iWorkingIndex].InRearPosition;
	END_IF
	IF bCylinderCheck THEN
		uiExecutingStep:=2500;
	ELSE
		tonTimeOut(IN:=TRUE, PT:=T#15S);
		IF tonTimeOut.Q THEN
			_Abort := TRUE;
			uiResumeStep := uiExecutingStep;
			strStatus := M_FormatManagedStatus(
				AlarmId := GVL_ErrorCode.GC_ALARM_ALC_OUTROBOT_REVERSE,
				InnerMessage := GVL_ErrorCode.GC_MSG_0052);
		END_IF
	END_IF

2500: // Next place? (修雙 clip 漏放 bug, 用 bPlacedA/B 旗標)
	IF bSyncPlace THEN
		bPlacedA := TRUE;
		bPlacedB := TRUE;
	ELSIF iWorkingIndex = 0 THEN
		bPlacedA := TRUE;
	ELSE
		bPlacedB := TRUE;
	END_IF
	IF UseA AND NOT bPlacedA THEN
		iWorkingIndex := 0;
		uiExecutingStep := 2000;
	ELSIF UseB AND NOT bPlacedB THEN
		iWorkingIndex := 1;
		uiExecutingStep := 2000;
	ELSE
		uiExecutingStep := 2600;
	END_IF

2600: // Move conveyor a bit until box detected at conveyor stop
	IF bMotorMoveForward THEN
		bMoveConveyorForward:=TRUE;
		bMoveConveyorBackrward:=FALSE;
	ELSE
		bMoveConveyorForward:=FALSE;
		bMoveConveyorBackrward:=TRUE;
	END_IF
	tonTimeDelay(IN:=NOT SensorOnConveyor, PT:=T#1S);
	IF tonTimeDelay.Q THEN
		uiExecutingStep:=2700;
	ELSE
		tonTimeOut(IN:=TRUE, PT:=T#15S);
		IF tonTimeOut.Q THEN
			_Abort := TRUE;
			uiResumeStep := uiExecutingStep;
			strStatus := M_FormatManagedStatus(
				AlarmId := GVL_ErrorCode.GC_ALARM_ALC_OUTROBOT_REVERSE,
				InnerMessage := GVL_ErrorCode.GC_MSG_0081);
		END_IF
	END_IF

2700: // Stop motor
	bMoveConveyorForward:=FALSE;
	bMoveConveyorBackrward:=FALSE;
	ConveyorMotor.M_MotorStop();
	IF ConveyorMotor.InStopped THEN
		uiExecutingStep:=3000;
	END_IF

3000: // Finish
	bMoveConveyorForward:=FALSE;
	bMoveConveyorBackrward:=FALSE;
	_Executed:=TRUE;

END_CASE

IF NOT Execute THEN
	eState:=STATE_RESETTING;
END_IF
IF _Error THEN
	eState:=STATE_ERROR;
END_IF
IF _Abort THEN
	eSTATE:=STATE_ABORTING;
END_IF
IF _Executed THEN
	eSTATE:=STATE_Done;
END_IF
END_METHOD

METHOD  M_STATE_RESETTING
VAR_INPUT
END_VAR
Busy := TRUE;
Error := _Error;

// Timer 確保歸零
tonTimeOut(IN:=FALSE);
tonTimeDelay(IN:=FALSE);

CASE uiResettingStep OF

	0:
		IF __ISVALIDREF(ConveyorMotor) THEN
			ConveyorMotor.M_MotorStop();
		END_IF
		M_RecoveryAllObjects();
		uiResettingStep:=9999;

	9999:
		Done := FALSE;
		Busy := FALSE;
		_ResetCompleted:=TRUE;
END_CASE

IF _ResetCompleted THEN
	eSTATE:=STATE_DORMANT;
END_IF
END_METHOD

END_FUNCTION_BLOCK

// ---- Library/20_MachineUnits/22_AllocateArea/Service/FB_OutRobot_BoxMoveTurnTableToRoundBelt.TcPOU
FUNCTION_BLOCK FB_OutRobot_BoxMoveTurnTableToRoundBelt EXTENDS FB_ObjectBase_V2
VAR_INPUT
//    Execute    :BOOL;   // True : This prog will start.
//    Abort      :BOOL;   // True : This prog will be abort.
//    Reset      :BOOL;   // True : This prog will be reset.
//    ObjectName :STRING; // Set this fb name(About it's action)
	INPUT            			   : REFERENCE TO ST_InputTable;
	Cylinders					   : REFERENCE TO ARRAY[0..1] OF FB_Cylinder;
	Clips						   : REFERENCE TO ARRAY[0..1] OF FB_Cylinder;
	AutoMode_TurnTableToRoundBelt : st_AutoMode_ClampingBoxesJob;	
END_VAR

VAR_OUTPUT
//    Busy    :BOOL;        // True : This prog is running.
//    Done    :BOOL;        // True : Command has been executed.
//    Aborted :BOOL;        // True : This prog is aborted.
//    Error   :BOOL;        // True : This prog has an error.
//    ErrorID :UINT;       // Output ErrorID
//    Status  :T_MaxString; // Output this prog status by string(255bytes)
END_VAR

VAR
//    eState :E_MethodStatus_Basic;
//	uiExecutingStep : UDINT; // This var is used to been controll STATE_EXECUTING process.
//	uiResettingStep : UDINT;
//	uiAbortingStep : UDINT;
//	_Executed :BOOL; // Executing process completed.
//	_Error : BOOL; // FB has an error.
//	_ResetCompleted : BOOL; // FB resetting completed.
//	_AbortCompleted : BOOL; // FB aborting completed.
	//_Abort		: BOOL;
	strStatus	: STRING;
	uiResumeStep : UINT;
	tonTimeOut   :TON;
	tonTimeDelay   :TON;
	iWorkingIndex : INT;
	_UniqueErrorCode :STRING;	
	PickingPos	: ARRAY[0..1] OF ST_PositionTable;
	PlacingPos  : ARRAY[0..1] OF ST_PositionTable;
	bSyncPick	: BOOL;
	bSyncPlace	: BOOL;	
	UseA	: BOOL;
	UseB	: BOOL;
END_VAR

A00_BasicUnits();
SUPER^.A10_StateControl();

ACTION A00_BasicUnits:
tonTimeOut(PT:=T#15S);
tonTimeDelay(PT:=T#1.5s);
END_ACTION

METHOD GetModelState
VAR_OUTPUT
    xDone    :BOOL;
    xBusy    :BOOL;
    xError   :BOOL;
    xAborted :BOOL;
    iErrorID :UDINT;
	UniqueErrorCode : STRING;
END_VAR
xDone    := Done;
xBusy    := Busy;
xError   := Error;
xAborted := Abort;
iErrorID := ErrorID;
UniqueErrorCode := THIS^.UniqueErrorCode;
END_METHOD

METHOD GetName : STRING
GetName := ObjectName;
END_METHOD

METHOD PRIVATE M_CheckCommand : BOOL
VAR_INPUT
END_VAR

M_CheckCommand := true;
END_METHOD

METHOD PRIVATE M_GetWorkingConditions : BOOL
VAR_INPUT
END_VAR
//For rare box move , Boxes must place on same position , therefor only work with TargetPosition of ClipA

IF AutoMode_TurnTableToRoundBelt.ClampingInfo.UseClibA THEN
	PickingPos[0] :=FUN_GetPositionTableData('R',1,0);
	PlacingPos[0] :=FUN_GetPositionTableData('A',5,0);
	UseA := TRUE;
END_IF

IF AutoMode_TurnTableToRoundBelt.ClampingInfo.UseClibB THEN
	PickingPos[1] :=FUN_GetPositionTableData('R',2,1);
	PlacingPos[1] :=FUN_GetPositionTableData('A',6,1);
	UseB :=TRUE;
END_IF

IF PlacingPos[0].X_Pos =PlacingPos[1].X_Pos AND PlacingPos[0].Y_Pos = PlacingPos[1].Y_Pos AND UseA AND UseB THEN
		bSyncPlace:=TRUE;
	ELSE
		bSyncPlace:=FALSE;	
END_IF
IF PickingPos[0].X_Pos =PickingPos[1].X_Pos AND PickingPos[0].Y_Pos = PickingPos[1].Y_Pos AND UseA AND UseB THEN
		bSyncPick:=TRUE;
	ELSE
		bSyncPick:=FALSE;	
END_IF
END_METHOD

METHOD PRIVATE M_RecoveryAllObjects : BOOL
VAR_INPUT
END_VAR
VAR 
	i : INT;
END_VAR
FOR i:=0 TO 1 DO
	IF Clips[i].xError THEN
		Clips[i].M_Reset();
		ELSE
		Clips[i].M_Retract();		
	END_IF
	IF Cylinders[i].xError THEN
	Cylinders[i].M_Reset();	
	ELSE
	Cylinders[i].M_Retract();	
	END_IF
END_FOR

IF arAxisCtrl_gb[AxisNo.OutRobot_X].Admin.Axis.Status.Error THEN

	arAxisCtrl_gb[AxisNo.OutRobot_X].Admin.ClearError:= TRUE;
ELSE
	arAxisCtrl_gb[AxisNo.OutRobot_X].Admin.ClearError:= FALSE;
END_IF

IF arAxisCtrl_gb[AxisNo.OutRobot_Y].Admin.Axis.Status.Error THEN

	arAxisCtrl_gb[AxisNo.OutRobot_Y].Admin.ClearError:= TRUE;
ELSE
	arAxisCtrl_gb[AxisNo.OutRobot_Y].Admin.ClearError:= FALSE;
END_IF
END_METHOD

METHOD  M_STATE_ABORTED
VAR_INPUT
END_VAR
ERROR :=TRUE;
Busy    := FALSE;
Aborted := TRUE;
Status := strStatus;

IF NOT Execute THEN
	eSTATE:=STATE_RESETTING;
END_IF

IF Execute AND Reset THEN
//	uiExecutingStep :=uiResumeStep;
	eSTATE:=STATE_EXECUTING;
END_IF
END_METHOD

METHOD  M_STATE_ABORTING
VAR_INPUT
END_VAR
VAR
	
i : int;
	bCylinderCheck: BOOL;
END_VAR
CASE uiAbortingStep OF
	0 :
		bCylinderCheck:=TRUE;
		FOR i :=0 TO 1 DO		
	    	Cylinders[i].M_Reset();
			Cylinders[i].M_Retract();
			bCylinderCheck:=bCylinderCheck AND Cylinders[i].InRearPosition;	
		END_FOR
		IF bCylinderCheck THEN		
			uiAbortingStep:=9999;
		END_IF
	
	9999:	_AbortCompleted:=TRUE;
END_CASE

IF _AbortCompleted THEN	
	eSTATE :=STATE_ABORTED;
END_IF
END_METHOD

METHOD  M_STATE_DONE
VAR_INPUT
END_VAR
Busy 	:= FALSE;
Done	:=TRUE;

IF NOT Execute THEN
	eSTATE:=STATE_RESETTING;
END_IF
END_METHOD

METHOD  M_STATE_DORMANT
VAR_INPUT
END_VAR
Busy            := FALSE;
Done            := FALSE;
Aborted         := FALSE;
Error           := FALSE;
ErrorID         := 0;
Status          := '';
_ResetCompleted := FALSE;
_Error          := FALSE;
_Executed       := FALSE;
strStatus :='FB_OutRobot_BoxMoveTurnTableToRoundBelt: No Error';
uiExecutingStep :=uiResettingStep :=uiResumeStep :=0;
tonTimeOut.IN :=TRUE;
_UniqueErrorCode:='0';
iWorkingIndex :=0;
bSyncPick :=FALSE;
bSyncPlace := FALSE;
UseA := FALSE;
UseB :=FALSE;

IF Execute THEN
	eSTATE:=STATE_EXECUTING;
END_IF
END_METHOD

METHOD  M_STATE_ERROR
VAR_INPUT
END_VAR
ERROR   :=TRUE;
Busy	:=FALSE;
Status := strStatus;
IF NOT Execute THEN	
eSTATE:=STATE_RESETTING;
END_IF
END_METHOD

METHOD  M_STATE_EXECUTING
VAR_INPUT
END_VAR
VAR_INST
	

END_VAR

VAR
	bCylinderCheck : BOOL := TRUE;
END_VAR
Busy :=TRUE;

CASE uiExecutingStep OF
	

0: //Idle
	tonTimeDelay.IN :=FALSE;
	tonTimeOut.IN := FALSE;
	iWorkingIndex :=0;	
	M_GetWorkingConditions();
	M_RecoveryAllObjects();
	uiExecutingStep := 100;
	
100: //Check command
	IF M_CheckCommand()THEN	
		uiExecutingStep:=200;
	END_IF
	
200: // Check  boxes on turntable

	IF (UseA AND NOT INPUT.bTurnTable_R1Detect_Sensor) OR (UseB AND NOT INPUT.bTurnTable_R2Detect_Sensor) THEN
		_Error:=TRUE;
		strStatus :='FB_OutRobot_BoxMoveTurnTableToRoundBelt Step 200: Box Not on Turntable';
	ELSE
		IF UseA THEN
			iWorkingIndex :=0;
		ELSE
			iWorkingIndex :=1;	
		END_IF
		
		uiExecutingStep:=1000;	
	END_IF

	
1000: 
	// Move OutRobot to First clip picking	
	 	 
	arAxisCtrl_gb[AxisNo.OutRobot_X].PosMode.Position := PickingPos[iWorkingIndex].X_Pos;		
	arAxisCtrl_gb[AxisNo.OutRobot_Y].PosMode.Position := PickingPos[iWorkingIndex].Y_Pos;	
	uiExecutingStep:=1100;
		// todo : Check axes is moving
1100:
	// Check outRobot arrived
	IF		(arAxisStatus_gb[AxisNo.OutRobot_X].Admin._OpModeAck = ModePosAbs AND arAxisStatus_gb[AxisNo.OutRobot_X].Admin.CmdDone) 
	AND (arAxisStatus_gb[AxisNo.OutRobot_Y].Admin._OpModeAck = ModePosAbs AND arAxisStatus_gb[AxisNo.OutRobot_Y].Admin.CmdDone) 
	THEN
		tonTimeOut.IN := FALSE;
		uiExecutingStep:=1200;
	END_IF	
	tonTimeOut.IN := TRUE;
	IF tonTimeOut.Q THEN
		tonTimeOut.IN := FALSE;
		_Error :=TRUE;
		strStatus :='FB_OutRobot_BoxMoveTurnTableToRoundBelt Step 1100: Robot move to picking position timeout';
	END_IF
	
1200: //Clip Down Pick	  
	bCylinderCheck := TRUE;
	Cylinders[iWorkingIndex].M_Extend();
	bCylinderCheck := Cylinders[iWorkingIndex].InFrontPosition AND bCylinderCheck;
	IF bSyncPick THEN
		Cylinders[1].M_Extend();
		bCylinderCheck := Cylinders[1].InFrontPosition AND bCylinderCheck;
	END_IF	
	 
	IF bCylinderCheck THEN
		tonTimeOut.IN := FALSE;
		uiExecutingStep:=1300;
	END_IF 
	tonTimeOut.IN := TRUE;
	IF tonTimeOut.Q THEN
		tonTimeOut.IN := FALSE;
		_Abort :=TRUE;
		strStatus :='FB_OutRobot_BoxMoveTurnTableToRoundBelt Step 1200: Cylinder pick down timeout';
	END_IF
	
1300: // Clip close Pick
	bCylinderCheck := TRUE;
	Clips[iWorkingIndex].M_Extend();
	bCylinderCheck := Clips[iWorkingIndex].InFrontPosition AND bCylinderCheck;
	IF bSyncPick THEN
		Clips[1].M_Extend();
		bCylinderCheck := Clips[1].InFrontPosition AND bCylinderCheck;
	END_IF	
	 
	IF bCylinderCheck THEN
		tonTimeOut.IN := FALSE;
		uiExecutingStep:=1400;
	END_IF 
	
		tonTimeOut.IN := TRUE;
	IF tonTimeOut.Q THEN
		tonTimeOut.IN := FALSE;
		_Abort :=TRUE;
		strStatus :='FB_OutRobot_BoxMoveTurnTableToRoundBelt Step 1300: clip pick close timeout';
	END_IF
	
1400: // Clip Up Pick
	bCylinderCheck := TRUE;
	Cylinders[iWorkingIndex].M_Retract();
	bCylinderCheck := Cylinders[iWorkingIndex].InRearPosition AND bCylinderCheck;
	IF bSyncPick THEN
		Cylinders[1].M_Retract();
		bCylinderCheck := Cylinders[1].InRearPosition AND bCylinderCheck;
	END_IF	
	 
	IF bCylinderCheck THEN
		tonTimeOut.IN := FALSE;
		uiExecutingStep:=1500;
	END_IF 
	
		tonTimeOut.IN := TRUE;
	IF tonTimeOut.Q THEN
		tonTimeOut.IN := FALSE;
		_Abort :=TRUE;
		strStatus :='FB_OutRobot_BoxMoveTurnTableToRoundBelt Step 1400: cylinder pick up timeout';
	END_IF
	  
1500: // If Next pick
	  IF iWorkingIndex>=1 OR bSyncPick OR NOT UseB THEN
		//Go to placing step
			IF UseA THEN
				iWorkingIndex:=0;
			ELSE
				iWorkingIndex:=1;	
			END_IF
			uiExecutingStep:=1600;
		ELSE
			iWorkingIndex :=iWorkingIndex +1;
			uiExecutingStep:=1000;	
	  END_IF
	  
1600: // Check box
		
	IF (UseA AND  INPUT.bTurnTable_R1Detect_Sensor) OR (UseB AND  INPUT.bTurnTable_R2Detect_Sensor) THEN
		
		//
	ELSE
		tonTimeOut.IN := FALSE;
		uiExecutingStep:=2000;
	END_IF
		tonTimeOut.IN := TRUE;
	IF tonTimeOut.Q THEN
		tonTimeOut.IN := FALSE;
		_Error :=TRUE;
		strStatus :='FB_OutRobot_BoxMoveTurnTableToRoundBelt Step 1600: Box still on Turntable';
	END_IF

2000: // Move to Placing pos	 
	 arAxisCtrl_gb[AxisNo.OutRobot_X].PosMode.Position := PlacingPos[iWorkingIndex].X_Pos;		
	 arAxisCtrl_gb[AxisNo.OutRobot_Y].PosMode.Position := PlacingPos[iWorkingIndex].Y_Pos;	
	 uiExecutingStep:=2100;

2100: // Waiting outRobot move to placing pos	 	
	 IF	(arAxisStatus_gb[AxisNo.OutRobot_X].Admin._OpModeAck = ModePosAbs AND arAxisStatus_gb[AxisNo.OutRobot_X].Admin.CmdDone) 
	AND (arAxisStatus_gb[AxisNo.OutRobot_Y].Admin._OpModeAck = ModePosAbs AND arAxisStatus_gb[AxisNo.OutRobot_Y].Admin.CmdDone)
	AND  tonTimeDelay.Q
	THEN		
		tonTimeOut.IN := FALSE;
		uiExecutingStep:=2200;
	END_IF	

		tonTimeOut.IN := TRUE;
	IF tonTimeOut.Q THEN
		tonTimeOut.IN := FALSE;
		_Error :=TRUE;
		strStatus :='FB_OutRobot_BoxMoveTurnTableToRoundBelt Step 2100: robot move to placing position timeout';
	END_IF


2200: //Cllp Down place
	bCylinderCheck := TRUE;
	Cylinders[iWorkingIndex].M_Extend();
	bCylinderCheck := Cylinders[iWorkingIndex].InFrontPosition AND bCylinderCheck;
	IF bSyncPlace THEN
		Cylinders[1].M_Extend();
		bCylinderCheck := Cylinders[1].InFrontPosition AND bCylinderCheck;
	END_IF	
	 
	IF bCylinderCheck THEN
		tonTimeOut.IN := FALSE;
		uiExecutingStep:=2300;
	END_IF 
		tonTimeOut.IN := TRUE;
	IF tonTimeOut.Q THEN
		tonTimeOut.IN := FALSE;
		_Abort :=TRUE;
		strStatus :='FB_OutRobot_BoxMoveTurnTableToRoundBelt Step 2200: Cylinder place down timeout';
	END_IF
	
2300: // Clip open Place
	bCylinderCheck := TRUE;
	Clips[iWorkingIndex].M_Retract();
	bCylinderCheck := Clips[iWorkingIndex].InRearPosition AND bCylinderCheck;
	IF bSyncPlace THEN
		Clips[1].M_Retract();
		bCylinderCheck := Clips[1].InRearPosition AND bCylinderCheck;
	END_IF	
	 
	IF bCylinderCheck THEN
		tonTimeOut.IN := FALSE;
		uiExecutingStep:=2400;
	END_IF 
	  
		tonTimeOut.IN := TRUE;
	IF tonTimeOut.Q THEN
		tonTimeOut.IN := FALSE;
		_Abort :=TRUE;
		strStatus :='FB_OutRobot_BoxMoveTurnTableToRoundBelt Step 2300: clip place open timeout';
	END_IF
	  
2400: // Clip up Placing
	bCylinderCheck := TRUE;
	Cylinders[iWorkingIndex].M_Retract();
	bCylinderCheck := Cylinders[iWorkingIndex].InRearPosition AND bCylinderCheck;
	IF bSyncPlace THEN
		Cylinders[1].M_Retract();
		bCylinderCheck := Cylinders[1].InRearPosition AND bCylinderCheck;
	END_IF	
	 
	IF bCylinderCheck THEN
		tonTimeOut.IN := FALSE;
		uiExecutingStep:=2500;
	END_IF 
		tonTimeOut.IN := TRUE;
	IF tonTimeOut.Q THEN
		tonTimeOut.IN := FALSE;
		_Abort :=TRUE;
		strStatus :='FB_OutRobot_BoxMoveTurnTableToRoundBelt Step 2400: cylinder place up timeout';
	END_IF
	
2500: // If Next place
	IF iWorkingIndex>=1 OR bSyncPlace OR NOT UseB THEN
		uiExecutingStep:=2600;
		// Finish
	ELSE	
		iWorkingIndex := iWorkingIndex+1;
	  	uiExecutingStep:=2000;
	END_IF
	
2600: // Finish	
	_Executed:=TRUE;
	
END_CASE
	
IF NOT Execute THEN
	eState:=STATE_RESETTING;
END_IF
IF _Error THEN
	eState:=STATE_ERROR;
END_IF
IF _Abort THEN
	eSTATE:=STATE_ABORTING;
END_IF
IF _Executed THEN
	eSTATE:=STATE_Done;
END_IF
END_METHOD

METHOD  M_STATE_RESETTING
VAR_INPUT
END_VAR
Busy := TRUE;
Error := _Error;


CASE uiResettingStep OF

	0:
		M_RecoveryAllObjects();
		uiResettingStep:=9999;


	9999:
		Done := FALSE;
		Busy := FALSE;
		_ResetCompleted:=TRUE;
END_CASE
IF _ResetCompleted THEN
	eSTATE:=STATE_DORMANT;
END_IF
END_METHOD

END_FUNCTION_BLOCK

// ---- Library/20_MachineUnits/22_AllocateArea/Service/FB_SameSizeCVCamera.TcPOU
FUNCTION_BLOCK FB_SameSizeCVCamera EXTENDS FB_ActionBasic
VAR_INPUT
    xExecute    : BOOL;
    xAbort      : BOOL;
	xReset		: BOOL;
    Cylinder 	: REFERENCE TO UNI_CylinderList;
    TimeOut  	: LREAL := 600; // Unit : s
	Input		: ST_InputTable;
	OutPut		: ST_OutputTable;
	Motor		: REFERENCE to UNI_MotorList;
	BoxCameraDone :BOOL;
END_VAR	
VAR_OUTPUT
    xAborted : BOOL;
    iErrorID : INT;
    ErrorMsg : STRING;
	UseBoxCamera	:BOOL;
END_VAR
VAR
    StateBehaviour   : CBML.ETrigATo;
    CurrentPosition : ST_PositionTable;
	uiCyclicStep    : UINT := 0;
	TON_DelaySensor	:TON;
	TON_TimeOut		:TON;
	TON_ArriviedTimeOut :TON ;
	TON_CameraTimeOut	:TON;
	TON_ConveyorTimeOut	:TON;
	Reset_Rtrig 	:R_TRIG;
	TON_SameSizeBoxDetect1_Delay :TON;
	fbExecuteEdgeDetect :FB_EdgeDetect;
	// ========== Resume 續做機制 ==========
	uiResumeStep	: UINT := 0;		// 錯誤發生時記錄的步驟，供續做使用
	bResumeEnabled	: BOOL := FALSE;	// 續做模式啟用旗標
END_VAR

THIS^.IBehaviourModel := StateBehaviour;

StateBehaviour(xExecute := xExecute,
              xAbort := xAbort OR fbExecuteEdgeDetect.xFallingEdge,
              udiTimeOut := LREAL_TO_UDINT( TimeOut*1000000),
              xDone => xDone,
              xBusy => xBusy,
              xError => xError,
              xAborted => xAborted);

fbExecuteEdgeDetect(xInput :=xExecute);

iErrorID := StateBehaviour._model.iErrorID;
ErrorMsg := M_GetErrorMsg(xErrorID := iErrorID);

Reset_Rtrig(CLK:= xReset);
IF Reset_Rtrig.Q THEN
	StateBehaviour.ResetModel(xCommit:=xReset);
END_IF

A00_BaseUnits();

ACTION A00_BaseUnits:
TON_DelaySensor(PT:= T#1S);
TON_TimeOut(PT := T#20S);
TON_ArriviedTimeOut(PT:= T#60S);
TON_CameraTimeOut(PT:=T#600S);
TON_ConveyorTimeOut(PT:=T#60S);
TON_SameSizeBoxDetect1_Delay(PT:=T#3S);
TON_SameSizeBoxDetect1_Delay.IN :=Input.bSameSizeCV_BoxDetect1_Sensor AND Motor.List.TransmitSameSideCV.InForWard;
END_ACTION

METHOD CleanupAction
VAR_INPUT
    xAbortProposed : BOOL;
    iErrorIDProposed: INT;
END_VAR
VAR_OUTPUT
    xComplete : BOOL := TRUE;
    xAbort: BOOL := xAbortProposed;
 	iErrorID : INT := iErrorIDProposed;
END_VAR
xComplete := FALSE;

// ============================================================
// Resume 機制：保存當前步驟供後續 Resume 使用
// ============================================================
IF uiResumeStep = 0 THEN
	uiResumeStep := uiCyclicStep;
END_IF

// 清除所有 Timer
TON_DelaySensor.IN 		:= FALSE;
TON_TimeOut.IN 			:= FALSE;
TON_ArriviedTimeOut.IN 	:= FALSE;
TON_CameraTimeOut.IN 	:= FALSE;
TON_ConveyorTimeOut.IN 	:= FALSE;

// 重置輸出信號
UseBoxCamera 	:= FALSE;
BoxCameraDone 	:= FALSE;

// 機械復位到安全狀態
IF NOT xExecute THEN
	Cylinder.List.fbSameSizeCV_Block1.M_Retract();
	Cylinder.List.fbSameSizeCV_Block2.M_Retract();
	Cylinder.List.fbTransmitCV_CamaraHoriz.M_Retract();
END_IF
Cylinder.List.fbSameSizeCV_Press1.M_Retract();
//Cylinder.List.fbSameSizeCV_Press2.M_Retract();
Motor.List.TransmitSameSideCV.M_MotorStop();

// 等待機械復位完成
IF NOT xExecute THEN
	IF Cylinder.List.fbSameSizeCV_Block1.InRearPosition AND
	   Cylinder.List.fbSameSizeCV_Block2.InRearPosition AND
	   Cylinder.List.fbSameSizeCV_Press1.InRearPosition AND
	   //Cylinder.List.fbSameSizeCV_Press2.InRearPosition AND
	   Cylinder.List.fbTransmitCV_CamaraHoriz.InRearPosition AND
	   Motor.List.TransmitSameSideCV.InStopped THEN
		xComplete := TRUE;
	END_IF
ELSE
	IF  Cylinder.List.fbSameSizeCV_Press1.InRearPosition AND
	   //Cylinder.List.fbSameSizeCV_Press2.InRearPosition AND
	   Motor.List.TransmitSameSideCV.InStopped THEN
		xComplete := TRUE;
	END_IF
END_IF
END_METHOD

METHOD CyclicAction
VAR_INPUT
    itfTimingController : CBML.ITimingController;
END_VAR
VAR_OUTPUT
    xComplete : BOOL := TRUE;
    iErrorID : INT := 0;
END_VAR
VAR_INST
	bMoveConveyorForward:BOOL;
END_VAR
xComplete := FALSE;
IF bMoveConveyorForward THEN
	IF NOT Motor.List.TransmitSameSideCV.InBackWard THEN
		Motor.List.TransmitSameSideCV.M_MoveForward();
	END_IF
END_IF

CASE uiCyclicStep OF
	0:	// 初始化
		bMoveConveyorForward:=FALSE;
		uiCyclicStep :=1000;
		
	1000:	// 擋第一個盒子
		TON_TimeOut.IN:=TRUE;
		Cylinder.List.fbSameSizeCV_Block1.M_Extend();
		Cylinder.List.fbTransmitCV_CamaraHoriz.M_Retract();
		IF Cylinder.List.fbSameSizeCV_Block1.InFrontPosition AND
			Cylinder.List.fbTransmitCV_CamaraHoriz.InRearPosition THEN
			TON_TimeOut.IN:=FALSE;
			uiCyclicStep :=1050;
		END_IF
		IF TON_TimeOut.Q THEN
			uiResumeStep := uiCyclicStep;
			iErrorID := 7;
		END_IF

	1050:	// 馬達前進
		TON_ConveyorTimeOut.IN:=TRUE;
		bMoveConveyorForward:=TRUE;
		Cylinder.List.fbSameSizeCV_Press2.M_Retract();
		IF Motor.List.TransmitSameSideCV.InForWard AND
			Cylinder.List.fbSameSizeCV_Press2.InRearPosition THEN
			TON_ConveyorTimeOut.IN:= FALSE;
			uiCyclicStep :=1100;
		END_IF
		IF TON_ConveyorTimeOut.Q THEN
			uiResumeStep := uiCyclicStep;
			iErrorID := 7;
		END_IF

	1100:	// 檢查盒子到達擋塊
		TON_ArriviedTimeOut.IN:=TRUE;
		TON_DelaySensor.IN:=Input.bSameSizeCV_BoxDetect2_Sensor;
		IF TON_DelaySensor.Q THEN
			TON_DelaySensor.IN :=FALSE;
			TON_ArriviedTimeOut.IN :=FALSE;
			Cylinder.List.fbSameSizeCV_Press2.M_Extend();
			bMoveConveyorForward:=FALSE;
			Motor.List.TransmitSameSideCV.M_MotorStop();
			uiCyclicStep :=1200;
		END_IF
		IF TON_ArriviedTimeOut.Q THEN
			uiResumeStep := uiCyclicStep;
			iErrorID := 8;
		END_IF

	1200:	// 發送拍照請求 & 擋住第二個盒子
		TON_ConveyorTimeOut.IN:=TRUE;
		IF Cylinder.List.fbSameSizeCV_Press2.InFrontPosition AND
			Motor.List.TransmitSameSideCV.InStopped THEN
			TON_ConveyorTimeOut.IN:= FALSE;
			UseBoxCamera :=TRUE;
			uiCyclicStep :=1300;
		END_IF
		IF TON_ConveyorTimeOut.Q THEN
			uiResumeStep := uiCyclicStep;
			iErrorID := 9;
		END_IF

	1300:	// 等待 C# 拍照完成 (Camera 錯誤不可續做)
		TON_CameraTimeOut.IN:=TRUE;
		IF BoxCameraDone THEN
			TON_CameraTimeOut.IN :=FALSE;
			Cylinder.List.fbSameSizeCV_Block1.M_Retract();
			bMoveConveyorForward:=TRUE;
			uiCyclicStep :=1400;
		END_IF
		IF TON_CameraTimeOut.Q THEN
			uiResumeStep := uiCyclicStep;
			iErrorID :=10;
		END_IF

	1400:	// 盒子通過 Detect1 感測器
		TON_TimeOut.IN :=TRUE;
		IF Input.bSameSizeCV_BoxDetect1_Sensor THEN
			TON_TimeOut.IN :=FALSE;
			uiCyclicStep :=1500;
		END_IF
		IF TON_TimeOut.Q THEN
			uiResumeStep := uiCyclicStep;
			iErrorID :=11;
		END_IF

	1500:	// 離開感測器後停止馬達
		TON_DelaySensor.IN :=TRUE;
		IF NOT Input.bSameSizeCV_BoxDetect1_Sensor THEN
			TON_DelaySensor.IN :=FALSE;
			bMoveConveyorForward:=FALSE;
			Motor.List.TransmitSameSideCV.M_MotorStop();
			uiCyclicStep :=1600;
		END_IF
		IF TON_DelaySensor.Q THEN 
			TON_DelaySensor.IN:=FALSE;
			bMoveConveyorForward:=FALSE;
			Motor.List.TransmitSameSideCV.M_MotorStop();
			uiCyclicStep :=1600;
		END_IF
	
	1600:	// 等待馬達停止
		IF Motor.List.TransmitSameSideCV.InStopped THEN
			xComplete :=TRUE;
		END_IF

END_CASE

IF TON_SameSizeBoxDetect1_Delay.Q THEN
	iErrorID := 20;
END_IF
END_METHOD

METHOD ExitAction
VAR_INPUT
    xAfterCleanup : BOOL;
    xInCopyCode : BOOL;
END_VAR
	uiCyclicStep    := 0;
	xAfterCleanup := true;
END_METHOD

METHOD M_GetErrorMsg : T_MaxString
VAR_INPUT
	xErrorID: INT;
END_VAR

VAR
	
END_VAR
CASE xErrorID OF
	0:
		M_GetErrorMsg := 'No Error';
	1:
		M_GetErrorMsg := 'FB_SameSizeCVCamera ErrorID 1: Action time out';
	2:
		M_GetErrorMsg := 'FB_SameSizeCVCamera ErrorID 2: Position Data invalid';
	3:
		M_GetErrorMsg := 'FB_SameSizeCVCamera ErrorID 3: Block1 cylinder not ready';
	4:
		M_GetErrorMsg := 'FB_SameSizeCVCamera ErrorID 4: Block2 cylinder not ready';
	5:
		M_GetErrorMsg := 'FB_SameSizeCVCamera ErrorID 5: Press1 cylinder not ready';
	6:
		M_GetErrorMsg := 'FB_SameSizeCVCamera ErrorID 6: Press2 cylinder not ready';
	7:
		M_GetErrorMsg := 'FB_SameSizeCVCamera ErrorID 7: CameraHoriz cylinder not ready';
	8:
		M_GetErrorMsg :='FB_SameSizeCVCamera ErrorID 8:  Box not arrived ';
	9:
		M_GetErrorMsg :='FB_SameSizeCVCamera ErrorID 9: Cylinder timeout';
	10:
		M_GetErrorMsg :='FB_SameSizeCVCamera ErrorID 10: box not arrived timeout';
	11:
		M_GetErrorMsg :='FB_SameSizeCVCamera ErrorID 11: Cylinder timeout';
	12:
		M_GetErrorMsg :='FB_SameSizeCVCamera ErrorID 12: C# send BoxCameraDone timeout';


	20:
		M_GetErrorMsg :='FB_SameSizeCVCamera ErrorID 20: SameSizeConveyor full box infront ';
END_CASE
END_METHOD

METHOD ResetAction
VAR_OUTPUT
    xComplete : BOOL := TRUE;
END_VAR
xComplete := FALSE;

// ============================================================
// Resume 機制判斷
// ------------------------------------------------------------
// 當錯誤發生後，操作員可選擇：
//   1. 保持 xExecute = TRUE 並按 Reset → Resume (從錯誤點繼續)
//   2. 先關閉 xExecute，再重新啟動 → 從頭開始
// ============================================================
bResumeEnabled := xExecute;

// 如果不是 Resume 模式，清除 Resume 步驟記錄
IF NOT bResumeEnabled THEN
	uiResumeStep := 0;
END_IF

// 清除所有 Timer
TON_DelaySensor.IN 		:= FALSE;
TON_TimeOut.IN 			:= FALSE;
TON_ArriviedTimeOut.IN 	:= FALSE;
TON_CameraTimeOut.IN 	:= FALSE;
TON_ConveyorTimeOut.IN 	:= FALSE;

xComplete := TRUE;
END_METHOD

METHOD StartAction
VAR_OUTPUT
    xComplete : BOOL := TRUE;
	iErrorID : INT := 0;
END_VAR
VAR
	bIsResumeMode : BOOL;	// 局部變數：記錄是否為 Resume 模式
END_VAR
xComplete := FALSE;

// 清除所有 Timer
TON_DelaySensor.IN 		:= FALSE;
TON_TimeOut.IN 			:= FALSE;
TON_ArriviedTimeOut.IN 	:= FALSE;
TON_CameraTimeOut.IN 	:= FALSE;
TON_ConveyorTimeOut.IN 	:= FALSE;

// ============================================================
// Resume 機制處理
// ------------------------------------------------------------
// 可 Resume 的錯誤: Error 7, 8, 9, 11 (氣缸/馬達/等待盒子)
// 不可 Resume 的錯誤: Error 10 (C# 拍照失敗), Error 20 (輸送帶滿載)
// ============================================================
bIsResumeMode := bResumeEnabled AND uiResumeStep > 0 AND uiResumeStep <> 1300;

IF bResumeEnabled AND uiResumeStep > 0 THEN
	IF uiResumeStep = 1300 THEN
		// Camera 錯誤：不可 Resume，強制從頭開始
		uiCyclicStep 	:= 0;
		UseBoxCamera 	:= FALSE;
		BoxCameraDone 	:= FALSE;
	ELSE
		// 其他錯誤：允許 Resume (人工已確認可繼續)
		uiCyclicStep := uiResumeStep;
	END_IF
	// 清除 Resume 旗標
	bResumeEnabled 	:= FALSE;
	uiResumeStep 	:= 0;
ELSE
	// 正常模式：從頭開始
	uiCyclicStep 	:= 0;
	UseBoxCamera 	:= FALSE;
	BoxCameraDone 	:= FALSE;
END_IF

// ============================================================
// 啟動前錯誤檢查
// ============================================================
IF TON_SameSizeBoxDetect1_Delay.Q THEN
	iErrorID := 20;
END_IF

IF Cylinder.List.fbSameSizeCV_Block1.xError THEN
	iErrorID := 3;
END_IF
IF Cylinder.List.fbSameSizeCV_Block2.xError THEN
	iErrorID := 4;
END_IF
IF Cylinder.List.fbSameSizeCV_Press1.xError THEN
	iErrorID := 5;
END_IF
IF Cylinder.List.fbSameSizeCV_Press2.xError THEN
	iErrorID := 6;
END_IF
IF Cylinder.List.fbTransmitCV_CamaraHoriz.xError THEN
	iErrorID := 7;
END_IF
IF Motor.List.TransmitSameSideCV.xError THEN
	iErrorID := 8;
END_IF

// 完成條件：Resume 模式直接完成，正常模式需檢查初始位置
IF bIsResumeMode OR
   (Cylinder.List.fbSameSizeCV_Block1.InRearPosition AND
    Motor.List.TransmitSameSideCV.InStopped) THEN
	xComplete := TRUE;
END_IF
END_METHOD

END_FUNCTION_BLOCK

// ---- Library/20_MachineUnits/22_AllocateArea/Service/FB_SameSizeCVCamera_Reverse.TcPOU
FUNCTION_BLOCK FB_SameSizeCVCamera_Reverse EXTENDS FB_ActionBasic
VAR_INPUT
    xExecute    : BOOL;
    xAbort      : BOOL;
	xReset		: BOOL;
    Cylinder 	: REFERENCE TO UNI_CylinderList;
    TimeOut  	: LREAL := 600; // Unit : s
	Input		: ST_InputTable;
	OutPut		: ST_OutputTable;
	Motor		: REFERENCE to UNI_MotorList;
	SameSizeCVRequest : REFERENCE TO ST_SameSizeCVRequest;	// Phase 2 仲裁:寫 bCamera_NeedBackward / bCamera_HoldStill
	BoxCameraDone :BOOL;
END_VAR
VAR_OUTPUT
    xAborted : BOOL;
    iErrorID : INT;
    ErrorMsg : STRING;
	UseBoxCamera	:BOOL;
END_VAR
VAR
    StateBehaviour   : CBML.ETrigATo;
    CurrentPosition : ST_PositionTable;
	uiCyclicStep    : UINT := 0;
	TON_DelaySensor	:TON;
	TON_TimeOut		:TON;
	TON_ArriviedTimeOut :TON ;
	TON_CameraTimeOut	:TON;
	TON_ConveyorTimeOut	:TON;
	Reset_Rtrig 	:R_TRIG;
	TON_SameSizeBoxDetect1_Delay :TON;
	fbExecuteEdgeDetect :FB_EdgeDetect;
	// ========== Resume 續做機制 ==========
	uiResumeStep	: UINT := 0;		// 錯誤發生時記錄的步驟，供續做使用
	bResumeEnabled	: BOOL := FALSE;	// 續做模式啟用旗標
END_VAR

THIS^.IBehaviourModel := StateBehaviour;

StateBehaviour(xExecute := xExecute,
              xAbort := xAbort OR fbExecuteEdgeDetect.xFallingEdge,
              udiTimeOut := LREAL_TO_UDINT( TimeOut*1000000),
              xDone => xDone,
              xBusy => xBusy,
              xError => xError,
              xAborted => xAborted);

fbExecuteEdgeDetect(xInput :=xExecute);

iErrorID := StateBehaviour._model.iErrorID;
ErrorMsg := M_GetErrorMsg(xErrorID := iErrorID);

Reset_Rtrig(CLK:= xReset);
IF Reset_Rtrig.Q THEN
	StateBehaviour.ResetModel(xCommit:=xReset);
END_IF

A00_BaseUnits();

ACTION A00_BaseUnits:
TON_DelaySensor(PT:= T#1S);
TON_TimeOut(PT := T#20S);
TON_ArriviedTimeOut(PT:= T#20S);	//等待盒子到位
TON_CameraTimeOut(PT:=T#30S);		// 拍照Timer
TON_ConveyorTimeOut(PT:=T#60S);
TON_SameSizeBoxDetect1_Delay(PT:=T#3S);
TON_SameSizeBoxDetect1_Delay.IN :=Input.bSameSizeCV_BoxDetect1_Sensor AND Motor.List.TransmitSameSideCV.InBackWard;
END_ACTION

METHOD CleanupAction
VAR_INPUT
    xAbortProposed : BOOL;
    iErrorIDProposed: INT;
END_VAR
VAR_OUTPUT
    xComplete : BOOL := TRUE;
    xAbort: BOOL := xAbortProposed;
 	iErrorID : INT := iErrorIDProposed;
END_VAR
xComplete := FALSE;

// ============================================================
// Resume 機制：保存當前步驟供後續 Resume 使用
// ============================================================
IF uiResumeStep = 0 THEN
	uiResumeStep := uiCyclicStep;
END_IF

// 清除所有 Timer
TON_DelaySensor.IN 		:= FALSE;
TON_TimeOut.IN 			:= FALSE;
TON_ArriviedTimeOut.IN 	:= FALSE;
TON_CameraTimeOut.IN 	:= FALSE;
TON_ConveyorTimeOut.IN 	:= FALSE;

// 重置輸出信號
UseBoxCamera 	:= FALSE;
BoxCameraDone 	:= FALSE;

// 機械復位到安全狀態
// Block1 / Press2 不由本 FB 管理 (上游 FB 持壓),cleanup 不縮回,避免盒子失壓往前溜
IF NOT xExecute THEN
	Cylinder.List.fbSameSizeCV_Block2.M_Retract();
	Cylinder.List.fbTransmitCV_CamaraHoriz.M_Retract();
END_IF

// Phase 2:cleanup 期間撤銷軌道請求 (xBusy gate),讓 arbiter 自然停 motor。
// xBusy 在 cleanup 期間 TRUE、idle FALSE,確保兩個 instance 不互相 stomp。
IF xBusy AND __ISVALIDREF(SameSizeCVRequest) THEN
	SameSizeCVRequest.bCamera_NeedBackward := FALSE;
	SameSizeCVRequest.bCamera_HoldStill    := FALSE;
END_IF

